*)
METHOD parse : BOOL
VAR_INPUT
	NMEAsentence : TNMEAsentence;
END_VAR
VAR_INST
	N 			: INT;
	msglen 		: INT;
	structlen	: INT;
	fieldtype	: BYTE;
	cbyte		: BYTE;
	fieldindex 	: INT;
	chkSumSentence  : USINT;
	chkSumCalc		: USINT;
	pbyte 			: POINTER TO BYTE; 
	ptypebyte		: POINTER TO BYTE;
	pbuffer 		: POINTER TO BYTE;
	pspointer		: POINTER TO STRING;
	buffer 			: TNMEAsentence;
END_VAR
parse := TRUE;
IF NOT getChkSumFromSentence(NMEAsentence, chkSumSentence) THEN
	parse := FALSE;
	RETURN;
END_IF

IF NOT calcChkSum(NMEASentence, chkSumCalc) THEN
	parse := FALSE;
	RETURN;
END_IF

IF chkSumCalc <> chkSumSentence THEN
	parse := FALSE;
	RETURN;
END_IF

msglen := len(NMEAsentence);
structlen := len(THIS^.sentenceStructure);

fieldindex := -1;

pbyte := ADR(NMEAsentence)+1;
ptypebyte := ADR(sentenceStructure);
pbuffer := ADR(buffer);

FOR N := 2 TO (msglen-2) DO
	cbyte := pbyte^;	
	
	CASE cbyte OF
		44, 42: // , and *
			pbuffer^ := 0;
			pbuffer := ADR(buffer); 
			pspointer := pbuffer;
			IF fieldindex = -1 THEN
				THIS^.header := pspointer^;
				fieldindex := 0;
			ELSE
				CASE ptypebyte^ OF
					73: // I
						THIS^.intFields[fieldindex] := STRING_TO_LINT(buffer);
						
					82: // R
						THIS^.realFields[fieldindex] := STRING_TO_LREAL(buffer);
						
					83: // S
					IF LEN(buffer) <= TNMEAstringsz THEN 
						THIS^.stringFields[fieldindex] := buffer;
					ELSE
						THIS^.stringFields[fieldindex] := '.';
					END_IF						
				END_CASE
				_incp(ptypebyte);
				fieldindex := fieldindex + 1;
				IF (structlen <= fieldindex) OR (cbyte = 42) THEN
					RETURN;
				END_IF
			END_IF
	ELSE
		pbuffer^ := cbyte;
		_incp(pbuffer);
 
	END_CASE	 
	_incp(pbyte);
 END_FOR
END_METHOD

(*
Purpose
=======
Set an string for field elements which are getting extracted. 
The position of a format char in the string is associated with the field number. 
The type of the field is given by the character

  I : Long Integer
  S : String(64)
  R : LReal
  . : Don't extract field
  
  Example:
  
  '..RR..I'
 
*)
METHOD setFieldsOfInterest : BOOL
VAR_INPUT
	Description : TNMEAStructDescription;
END_VAR
THIS^.sentenceStructure := Description;
END_METHOD

END_FUNCTION_BLOCK

// NMEA/NMEASentence
FUNCTION_BLOCK NMEASentence
VAR_INPUT
	
END_VAR
VAR
	formatString : FB_FormatString2;
	_dataOut : TNMEASentence;	
END_VAR

METHOD PROTECTED calcCheckSum : STRING
VAR_INPUT
	data : REFERENCE TO TNMEAsentence;	
END_VAR
VAR
	checksum : USINT;
	msglen : INT;
	N : INT;
	chksum : BYTE;
	char : BYTE; 
	pbyte : POINTER TO BYTE;
	x : BYTE;	
END_VAR
checksum := 0;
msglen := LEN(Data);
pbyte := ADR(data)+1;

FOR N := 2 TO msglen DO
	IF (pbyte^=42) THEN // Char *
		EXIT;
	ELSIF  (pbyte^=10) OR (pbyte^=13) THEN // Chars NL and CR
		EXIT;
	END_IF
	
	checksum := checksum XOR pbyte^;
	pbyte := pbyte + 1;
END_FOR

calcCheckSum :=  BYTE_TO_HEXSTR(In:= checksum, iPrecision:=2, bLoCase:=FALSE);
END_METHOD

PROPERTY DataOut : STRING
GET
DataOut := _dataout;
END_GET
END_PROPERTY

METHOD formatSentenceWith3Values : BOOL
VAR_INPUT
	NMEAType: REFERENCE TO T_MaxString;	
	Value1 	: LREAL;
	Value2 	: LREAL;
	Value3 	: LREAL;
END_VAR
VAR CONSTANT
		FORMATSTR 	: TNMEASentence := '%S,%.2F,%.2F,%.2F*  $0D$0A';
END_VAR
VAR
	checksum : STRING;
	datalen : INT;
END_VAR
formatString(pFormatString:=ADR(FORMATSTR), 
					arg1:=F_STRING(NMEAType), arg2:=F_LREAL(Value1), arg3:= F_LREAL(Value2), arg4:=F_LREAL(Value3), 
					pDstString:=ADR(_dataOut), nDstSize:=TO_UDINT(255)); 
					
		
checksum := calcCheckSum(data:=_dataout);
datalen := LEN(_dataout);


_dataout := REPLACE(_dataout,checksum, 2, datalen-3);
END_METHOD

END_FUNCTION_BLOCK

// NMEA/NMEA_TrawlLength
FUNCTION_BLOCK NMEA_TrawlLength EXTENDS NMEASentence
VAR_INPUT
	LengthSTBD 	: LREAL;
	LengthPORT 	: LREAL;
	LengthMID 	: LREAL;	
END_VAR
VAR CONSTANT
	NMEAType : T_MaxString := '@TAWWL';
END_VAR

SUPER^.formatSentenceWith3Values(NMEAType:= NMEAType, Value1:=LengthSTBD, Value2:=LengthPORT, Value3:=LengthMID);

END_FUNCTION_BLOCK

// NMEA/NMEA_TrawlSpeed
FUNCTION_BLOCK NMEA_TrawlSpeed EXTENDS NMEASentence
VAR_INPUT
	SpeedSTBD 	: LREAL;
	SpeedPORT 	: LREAL;
	SpeedMID 	: LREAL;	
END_VAR
VAR CONSTANT
	NMEAType : T_MaxString := '@TAWWS';
END_VAR

VAR_OUTPUT
END_VAR
VAR
END_VAR

SUPER^.formatSentenceWith3Values(NMEAType:= NMEAType, Value1:=SpeedSTBD, Value2:=SpeedPORT, Value3:=SpeedMID);

END_FUNCTION_BLOCK

// NMEA/NMEA_TrawlTension
FUNCTION_BLOCK NMEA_TrawlTension EXTENDS NMEASentence
VAR_INPUT
	TensionSTBD 	: LREAL;
	TensionPORT 	: LREAL;
	TensionMID 	: LREAL;	
END_VAR
VAR CONSTANT
	NMEAType : T_MaxString := '@TAWWT';
END_VAR

VAR_OUTPUT
END_VAR
VAR
END_VAR

SUPER^.formatSentenceWith3Values(NMEAType:= NMEAType, Value1:=TensionSTBD, Value2:=TensionPORT, Value3:=TensionMID);

END_FUNCTION_BLOCK

// NMEA/NMEATransmitter6021
FUNCTION_BLOCK NMEATransmitter6021
VAR_INPUT
	data 	: REFERENCE TO TNMEASentence;
	start   : BOOL;
END_VAR
VAR
	dataout AT %Q*  : ARRAY[0..97] OF BYTE;
	sword	AT %I*  : WORD;
	cword	AT %Q*  : WORD;
	_busy			: BOOL;
	state			: DINT;
	started			: BOOL;
END_VAR



CASE state OF
	0: 
		_busy := FALSE;
		IF NOT started THEN
			state := 100;
		ELSIF start THEN
			state := 10;
		END_IF
	10:
		_busy := TRUE;
		strncpy(ADR(dataout), ADR(data), TO_UINT(LEN(data)+1));
		cword := SHL(TO_UINT(len(data)), 8) OR (cword AND 16#0001);
		cword.0 := NOT cword.0;
		_busy := TRUE;
		state := 20;
		
	20:
		IF sword.0 THEN
			state := 0;
		END_IF
	
	100:
		_busy := TRUE;
		cword.2 := TRUE;	
		IF sword.2 AND NOT start THEN
			cword.2 := FALSE;
			started :=TRUE;
			state := 110; 
		END_IF	
		
	110: 
		cword := 0;
		IF NOT sword.2	THEN
			state := 0;
			_busy := FALSE;
		END_IF
END_CASE

PROPERTY Busy : BOOL
GET
Busy := _busy;
END_GET
END_PROPERTY

END_FUNCTION_BLOCK

// ObjectProtocols/V1/ProtoBase1ToN
(* 
Protocol Base Class 1:N
=======================

The class is class partially implementing a simple relation between objects of 1:N

This class has to be derived and can't be used out of the box. 

You have to take care of _noElements, _totalSize

*)

{attribute 'hide_all_locals'}
FUNCTION_BLOCK ABSTRACT ProtoBase1ToN IMPLEMENTS p7type.IProtoBase1ToN
VAR
	_noElements : DINT;
	_totalSize  : DINT;
END_VAR

METHOD attach : IProtoBase1ToN
VAR_INPUT
	Service : IProtoService;
END_VAR
VAR
	N	 		: DINT;
	_service	: IProtoService;
END_VAR

FOR N := 0 TO THIS^._totalSize-1 DO
	//We can't compare an Interface value returned from a method, which makes this 
	// necessary
	_service := getService(N);
	IF _service = Service THEN
		EXIT;
	ELSIF _service = 0 THEN
		setService(N, Service);
		_noElements := _noElements + 1;
		EXIT;
	END_IF
END_FOR

attach := THIS^;
END_METHOD

// This method has initialize _totalSize
METHOD FB_init : BOOL
VAR_INPUT
	bInitRetains : BOOL; // if TRUE, the retain variables are initialized (warm start / cold start)
	bInCopyCode : BOOL;  // if TRUE, the instance afterwards gets moved into the copy code (online change)
END_VAR
THIS^._totalSize := Parameters.ServicesPerMaster;

_noElements := 0;
END_METHOD

METHOD getNoServices : DINT
getNoServices := _noElements;
END_METHOD

// Overwrite this method
METHOD PROTECTED ABSTRACT getService : IProtoService
VAR_INPUT
	Index  : DINT;
END_VAR
END_METHOD

METHOD getServiceByIdx : IProtoService
VAR_INPUT
	Index  : DINT;
END_VAR
getServiceByIdx := getService(Index);
END_METHOD

METHOD isAttached : BOOL
VAR_INPUT
	Service : IProtoService;
END_VAR
VAR
	N : DINT;
	_service	: IProtoService;
END_VAR
isAttached := FALSE;
FOR N := 0 TO THIS^._totalSize-1 DO
	//We can't compare an Interface value returned from a method, which makes this 
	// necessary
	_service := getService(N);
	IF Service = _service THEN
		isAttached := TRUE;
		EXIT;
	ELSIF _service = 0 THEN
		EXIT;
	END_IF
END_FOR
END_METHOD

METHOD resetService : IProtoBase1ToN
VAR
	N 			: DINT;
	noElements 	: DINT;
END_VAR
FOR N := 0 TO THIS^._totalSize-1 DO
	setService(N, 0);
END_FOR

THIS^._noElements := 0;

resetService := THIS^;
END_METHOD

// Overwrite this method
METHOD PROTECTED ABSTRACT setService : IProtoBase1ToN
VAR_INPUT
	Index : DINT;
	Value : IProtoService;
END_VAR
END_METHOD

END_FUNCTION_BLOCK

// ObjectProtocols/V1/ProtoBaseNTo1
(* 
Protocol Base Class N:1
=======================

The class is class partially implementing a simple relation between objects of N:1. The 1 element is a master, which 
has to provide IProtoMasterSingleService to attach remote a Service by the service

This class has to be derived and can't be used out of the box. 

You have to take care of _noElements, _totalSize


*)

{attribute 'hide_all_locals'}
FUNCTION_BLOCK ABSTRACT ProtoBaseNTo1 IMPLEMENTS p7type.IProtoBaseNTo1
VAR
	_noElements : DINT;
	_totalSize  : DINT;
END_VAR

METHOD attach : IProtoBaseNTo1
VAR_INPUT
	Master	: IProtoMasterSingleService;
END_VAR
VAR
	N 		: DINT;
	_master : IProtoMasterSingleService;
END_VAR

FOR N := 0 TO THIS^._totalSize-1 DO
	_master := THIS^.getMaster(N);
	IF _master = Master THEN
		EXIT;
	ELSIF _master = 0 THEN
		setMaster(N, Master);
		Master.attach(THIS^);
		_noElements := _noElements + 1;
		EXIT;
	END_IF
END_FOR

attach := THIS^;
END_METHOD

// This method has initialize _totalSize
METHOD FB_init : BOOL
VAR_INPUT
	bInitRetains : BOOL; // if TRUE, the retain variables are initialized (warm start / cold start)
	bInCopyCode : BOOL;  // if TRUE, the instance afterwards gets moved into the copy code (online change)
END_VAR
THIS^._totalSize := Parameters.MastersPerService;

_noElements := 0;
END_METHOD

{attribute 'monitoring' := 'call'}
// Overwrite this method
METHOD PROTECTED ABSTRACT getMaster : IProtoMasterSingleService
VAR_INPUT
	Index  : DINT;
END_VAR
END_METHOD

METHOD getMasterByIdx : IProtoMasterSingleService
VAR_INPUT
	Index  : DINT;
END_VAR
	getMasterByIdx := getMaster(Index);
END_METHOD

METHOD getNoMasters : DINT
getNoMasters := THIS^._noElements;
END_METHOD

METHOD isAttached : BOOL
VAR_INPUT
	Master	: IProtoMasterSingleService;
END_VAR
VAR
	N : DINT;
	_master : IProtoMasterSingleService;
END_VAR
isAttached := FALSE;
FOR N := 0 TO THIS^._totalSize-1 DO
	_master := getMaster(N);
	IF Master = _master THEN
		isAttached := TRUE;
		EXIT;
	ELSIF _master = 0 THEN
		EXIT;
	END_IF
END_FOR
END_METHOD

METHOD resetServices : IProtoBaseNTo1
VAR
	N : DINT;
END_VAR
FOR N := 0 TO _totalSize-1 DO
	setMaster(N, 0);
END_FOR
_noElements := 0;

resetServices := THIS^;
END_METHOD

// Overwrite this method
METHOD PROTECTED setMaster : IProtoBaseNTo1
VAR_INPUT
	Index : DINT;
	Value : IProtoMasterSingleService;
END_VAR
END_METHOD

END_FUNCTION_BLOCK

// ObjectProtocols/V1/ProtoMasterSingleService

{attribute 'hide_all_locals'}
FUNCTION_BLOCK ProtoMasterSingleService IMPLEMENTS p7type.IProtoMasterSingleService
VAR
	service 			: IProtoService; 
END_VAR

METHOD attach : IProtoMasterSingleService
VAR_INPUT
	Service	: IProtoService;
END_VAR
THIS^.service := Service;

attach := THIS^;
END_METHOD

METHOD getService : IProtoService
getService := THIS^.service;
END_METHOD

END_FUNCTION_BLOCK

// OperationTime/DeviceOpTime
(* This utility class is counting optime for winches in hours
	Internaly the counter is of type TIME, but the output is of type UINT
*)
FUNCTION_BLOCK DeviceOpTime
VAR_INPUT
	Device : p7type.IP6OpState;
END_VAR
VAR PERSISTENT
	_optime : TIME;
END_VAR
VAR
	counter : OperationTimeCounter;
END_VAR

IF Device = 0 THEN
	RETURN;
END_IF

counter.update(
	active := Device.OpState = p7type.P6OpState.RUN,
	operationTime := _optime
);

{attribute 'monitoring' := 'call'}
{attribute 'TcRpcEnable'}
PROPERTY Optime : UDINT
GET
OpTime := TIME_TO_UDINT(_optime/UDINT#3600000);
END_GET
SET
_optime := UDINT_TO_TIME(Optime*UDINT#3600000);
END_SET
END_PROPERTY

END_FUNCTION_BLOCK

// OperationTime/OperationTimeCounter
// The class measures the active-time and adds it to the referenced operationTime. 
{attribute 'hide_all_locals'}
FUNCTION_BLOCK OperationTimeCounter
VAR
	_startTime 			: TIME;
	_state 				: OperationTimeSM;
	optime				: REFERENCE TO TIME;
END_VAR

METHOD reset : BOOL
THIS^.optime := T#0S;
END_METHOD

METHOD update : BOOL
VAR_INPUT
	active : BOOL;
	operationTime : REFERENCE TO TIME;
END_VAR
optime REF= operationTime;

CASE _state OF
	OperationTimeSM.IDLE:
		IF active THEN
			_state := OperationTimeSM.ACTIVE;
			_startTime := TIME();
		END_IF
			
	OperationTimeSM.ACTIVE:
		IF NOT active THEN
			operationTime := operationTime + (TIME() - _startTime);
			_state := OperationTimeSM.IDLE;
		ELSE
			_state := OperationTimeSM.ACTIVE;
			operationTime := operationTime + (TIME() - _startTime);
			_startTime := TIME();			
		END_IF
END_CASE
END_METHOD

END_FUNCTION_BLOCK

// ParameterManagment/AddParameter/AddParameterBool
FUNCTION_BLOCK AddParameterBool
VAR_INPUT
	parameterName : STRING := 'NoParameterNameSet'; //Parameter name to be displayed
	unit : STRING := ''; //SI units (m, kg, Nm, etc.)
	uploadParameter : BOOL := FALSE; //Update parameters to PLC
	downloadParameter : BOOL := FALSE; //Download parameters to HMI
END_VAR
VAR_OUTPUT
END_VAR
VAR_IN_OUT
	configMember : BOOL;
	parameterList : ParameterList;
END_VAR
VAR
	_init : BOOL := TRUE;
END_VAR

IF _init THEN
	_init := FALSE;
	parameterList.name := parameterName;
	parameterList.unit := unit;
END_IF

IF uploadParameter THEN
	configMember := parameterList.value.boolType;
END_IF

IF downloadParameter THEN
	parameterList.value.boolType := configMember;
END_IF

//Check status on parameter between config and parameter list
IF (parameterList.value.boolType = configMember)
THEN
	parameterList.status := 'Ok';
ELSE
	parameterList.status := 'Missmatch!';
END_IF

END_FUNCTION_BLOCK

// ParameterManagment/AddParameter/AddParameterInt
FUNCTION_BLOCK AddParameterInt
VAR_INPUT
	parameterName : STRING := 'NoParameterNameSet'; //Parameter name to be displayed
	unit : STRING := ''; //SI units (m, kg, Nm, etc.)
	uploadParameter : BOOL := FALSE; //Update parameters to PLC
	downloadParameter : BOOL := FALSE; //Download parameters to HMI
END_VAR
VAR_OUTPUT
END_VAR
VAR_IN_OUT
	configMember : INT;
	parameterList : ParameterList;
END_VAR
VAR
	_init : BOOL := TRUE;
END_VAR

IF _init THEN
	_init := FALSE;
	parameterList.name := parameterName;
	parameterList.unit := unit;
END_IF

IF uploadParameter THEN
	configMember := parameterList.value.intType;
END_IF

IF downloadParameter THEN
	parameterList.value.intType := configMember;
END_IF

//Check status on parameter between config and parameter list
IF (parameterList.value.intType = configMember)
THEN
	parameterList.status := 'Ok';
ELSE
	parameterList.status := 'Missmatch!';
END_IF

END_FUNCTION_BLOCK

// ParameterManagment/AddParameter/AddParameterLreal
FUNCTION_BLOCK AddParameterLreal
VAR_INPUT
	parameterName : STRING := 'NoParameterNameSet'; //Parameter name to be displayed
	unit : STRING := ''; //SI units (m, kg, Nm, etc.)
	uploadParameter : BOOL := FALSE; //Update parameters to PLC
	downloadParameter : BOOL := FALSE; //Download parameters to HMI
END_VAR
VAR_OUTPUT
END_VAR
VAR_IN_OUT
	configMember : LREAL;
	parameterList : ParameterList;
END_VAR
VAR
	_init : BOOL := TRUE;
END_VAR

IF _init THEN
	_init := FALSE;
	parameterList.name := parameterName;
	parameterList.unit := unit;
END_IF

IF uploadParameter THEN
	configMember := parameterList.value.lrealType;
END_IF

IF downloadParameter THEN
	parameterList.value.lrealType := configMember;
END_IF

//Check status on parameter between config and parameter list
IF (parameterList.value.lrealType = configMember)
THEN
	parameterList.status := 'Ok';
ELSE
	parameterList.status := 'Missmatch!';
END_IF

END_FUNCTION_BLOCK

// ParameterManagment/AddParameter/AddParameterStr
FUNCTION_BLOCK AddParameterStr
VAR_INPUT
	parameterName : STRING := 'NoParameterNameSet'; //Parameter name to be displayed
	unit : STRING := ''; //SI units (m, kg, Nm, etc.)
	uploadParameter : BOOL := FALSE; //Update parameters to PLC
	downloadParameter : BOOL := FALSE; //Download parameters to HMI
END_VAR
VAR_OUTPUT
END_VAR
VAR_IN_OUT
	configMember : STRING;
	parameterList : ParameterList;
END_VAR
VAR
	_init : BOOL := TRUE;
END_VAR

IF _init THEN
	_init := FALSE;
	parameterList.name := parameterName;
	parameterList.unit := unit;
END_IF

IF uploadParameter THEN
	configMember := parameterList.value.stringType;
END_IF

IF downloadParameter THEN
	parameterList.value.stringType := configMember;
END_IF

//Check status on parameter between config and parameter list
IF (parameterList.value.stringType = configMember)
THEN
	parameterList.status := 'Ok';
ELSE
	parameterList.status := 'Missmatch!';
END_IF

END_FUNCTION_BLOCK

// ParameterManagment/AddParameter/AddParameterTime
FUNCTION_BLOCK AddParameterTime
VAR_INPUT
	parameterName : STRING := 'NoParameterNameSet'; //Parameter name to be displayed
	unit : STRING := ''; //SI units (m, kg, Nm, etc.)
	uploadParameter : BOOL := FALSE; //Update parameters to PLC
	downloadParameter : BOOL := FALSE; //Download parameters to HMI
END_VAR
VAR_OUTPUT
END_VAR
VAR_IN_OUT
	configMember : TIME;
	parameterList : ParameterList;
END_VAR
VAR
	_init : BOOL := TRUE;
	_msPerSecond : LREAL := 1000.0;
END_VAR

IF _init THEN
	_init := FALSE;
	parameterList.name := parameterName;
	parameterList.unit := unit;
END_IF

IF uploadParameter THEN
	configMember := LREAL_TO_TIME(parameterList.value.lrealType * _msPerSecond);
END_IF

IF downloadParameter THEN
	parameterList.value.lrealType := TIME_TO_LREAL(configMember) / _msPerSecond;
END_IF

//Check status on parameter between config and parameter list
IF (parameterList.value.lrealType * _msPerSecond = TIME_TO_LREAL(configMember)) THEN
	parameterList.status := 'Ok';
ELSE
	parameterList.status := 'Missmatch!';
END_IF

END_FUNCTION_BLOCK

// PID/HTrawlController
(*
Purpose
=======
This is a 2 stage P-PI controller for trawling withg hydraulic winches.
This is the first version and only for documentations purposes in this lib. 

Features
========
#. This version has no stepped P controller for velocity
#. Anti Windup for the integrator
#. Symmetric processing to 0 of input values
#. Limiting output values 

Methods And Properties
======================
*)
{attribute 'hide_all_locals'}
FUNCTION_BLOCK HTrawlController;
VAR_INPUT
	config 				: REFERENCE TO p7type.ConfigTrawlController;
	Active 				: BOOL;		
	IsInRun				: BOOL;
	PayoutMode			: BOOL;
	Setpoint 			: LREAL;	// Length setpoint
	ProcessValueLen		: LREAL;	// Length process value
	ProcessValueVel		: LREAL;	// Velocity process value
	ProcessValueTension : LREAL;	// Tension process value 
	ProcessValueTorqueRel: LREAL;
	LimitVel			: LREAL;
	LimitTensionMax		: LREAL;
	LimitTensionMin		: LREAL;
	LimitTorqueRelMax	: LREAL;
	LimitTorqueRelMin	: LREAL;
	IntegratorPresetRel : LREAL;
	ReduceEnergyUsage	: BOOL;
	CycleTime			: LREAL;
END_VAR
VAR CONSTANT
	ALMOST_ZERO 		: LREAL := 1.0/60.0;
END_VAR
VAR
	startTrig 			: R_TRIG;
	_torqueOut 			: LREAL;
	Tc					: LREAL;
	errorLen			: LREAL;
	errorVel			: LREAL;
	deltaIt				: LREAL;
	tmp 				: LREAL;
	It					: LREAL;
	Pt					: LREAL;
	
	setpointVelocity		: LREAL;
	step				: DINT;
	velocityReduction   : LREAL;
	timerReducePower	: BOOL;
	statePos			: UINT;
	positionChange		: BOOL;
	offsetTension		: LREAL;
	pValueTension		: LREAL;
	pLimitTensionMax	: LREAL;
	pLimitTensionMin	: LREAL;
END_VAR

Tc := CycleTime;
//
// Process the position error
// 
errorLen :=  (SetPoint - ProcessValueLen);
 
(* Process deadband *)
IF Config.DeadbandLength > 0 THEN
	IF (ABS(errorLen) < (Config.DeadbandLength/2.0)) THEN
		errorLen := 0.0;
	ELSE 
		errorLen := errorLen - Signum(errorLen) * Config.DeadbandLength/2.0; 
	END_IF;
END_IF;

IF Active THEN
	// Initiatlize integrator for torque
	startTrig(CLK:=Active);
	IF startTrig.Q AND IsInRun THEN
		It := ProcessValueTorqueRel-0.5;
		step := 0;
	ELSIF startTrig.Q AND (NOT IsInRun)  THEN
		It :=  LIMIT(-0.5, IntegratorPresetRel-0.5, 0.5);
	END_IF
		
	IF ReduceEnergyUsage THEN 
		velocityReduction := 0.1;
	ELSE
		velocityReduction := 1;
	END_IF
	setpointVelocity := LIMIT(-LimitVel*velocityReduction ,errorLen*config.KpVelocity*velocityReduction, LimitVel*velocityReduction);
	//setpointVelocity := LIMIT(-LimitVel ,errorLen * config.KpVelocity, LimitVel);
	
	//
	// Tension controller -> Control velocity with torque
	//

	// The minus has to be used bc of torque has the opposite direction to velocity 
	errorVel := - (setpointVelocity - ProcessValueVel);	
	Pt := config.KpTorque * errorVel;
	
	
	IF ProcessValueVel <= (-LimitVel) THEN
		It := It - config.KiVelocityLimit;
		It := LIMIT(-0.5, It, 0.5);
		step := 2;
	ELSIF ProcessValueVel >= (LimitVel) THEN
		It := It + config.KiVelocityLimit;
		It := LIMIT(-0.5, It, 0.5);				
		step := 3;
	ELSIF (ProcessValueTension  < LimitTensionMin) THEN
		It := It + config.KiTensionLimit;
		It := LIMIT(-0.5, It, 0.5);
		step := 4;
	ELSIF (ProcessValueTension  > LimitTensionMax) AND (NOT PayoutMode) THEN
		It := It - config.KiTensionLimit;
		It := LIMIT(-0.5, It, 0.5);
		step := 5;
	ELSIF ABS(Config.KiTorque) <= 1E-100 THEN
		It :=  0.0;
		deltaIt := 0.0;
		step := 6;
	ELSE
		step := 1;
		// Start the check whether the new output would saturate and don't integrate when 
		// this is case
		deltaIt := errorVel * config.KiTorque * Tc;
		
		tmp := Pt + It + deltaIt;
		
		IF ABS(tmp) <= 0.5  THEN
			It := It + deltaIt;
		END_IF		
	END_IF

	
	_torqueOut := LIMIT(0, (Pt + It + 0.5), 1);	
ELSE
	_torqueOut := ProcessValueTorqueRel;// normalized to 1
END_IF;

{attribute 'TcRpcEnable'}
{attribute 'monitoring' := 'variable'}
PROPERTY ErrorPosition : LREAL
GET
ErrorPosition := errorLen;
END_GET
END_PROPERTY

{attribute 'TcRpcEnable'}
{attribute 'monitoring' := 'variable'}
PROPERTY ErrorVelocity : LREAL
GET
ErrorVelocity := errorVel;
END_GET
END_PROPERTY

{attribute 'TcRpcEnable'}
{attribute 'monitoring' := 'variable'}
PROPERTY Tension : LREAL
GET
Tension := TorqueOut;
END_GET
END_PROPERTY

PROPERTY TorqueOut : LREAL
GET
TorqueOut := _torqueOut;
END_GET
END_PROPERTY

END_FUNCTION_BLOCK

// PID/HTrawlController2
(*
Purpose
=======
This is a 2 stage P-PI controller for trawling withg hydraulic winches
This 2nd version is limit velocity via setpoint for the inner controller and
tension via limiting torqueRel. 

Features
========
#. This version has no stepped P controller for velocity
#. Anti Windup for the integrator
#. Symmetric processing to 0 of input values
#. Limiting output values 

Methods And Properties
======================
*)
{attribute 'hide_all_locals'}
FUNCTION_BLOCK HTrawlController2;
VAR_INPUT
	config 				: REFERENCE TO p7type.ConfigTrawlController;
	Active 				: BOOL;		
	IsInRun				: BOOL;
	PayoutMode			: BOOL;
	Setpoint 			: LREAL;	// Length setpoint
	ProcessValueLen		: LREAL;	// Length process value
	ProcessValueVel		: LREAL;	// Velocity process value
	ProcessValueTension : LREAL;	// Tension process value 
	ProcessValueTorqueRel: LREAL;
	LimitVel			: LREAL;
	LimitTensionMax		: LREAL;
	LimitTensionMin		: LREAL;
	LimitTorqueRelMax	: LREAL;
	LimitTorqueRelMin	: LREAL;
	IntegratorPresetRel : LREAL;
	ReduceEnergyUsage	: BOOL;
	CycleTime			: LREAL;
END_VAR
VAR CONSTANT
	ALMOST_ZERO 		: LREAL := 1.0/60.0;
END_VAR

VAR
	startTrig 			: R_TRIG;
	_torqueOut 			: LREAL;
	Tc					: LREAL;
	errorLen			: LREAL;
	errorVel			: LREAL;
	deltaIt				: LREAL;
	tmp 				: LREAL;
	It					: LREAL;
	Pt					: LREAL;
	
	setpointVelocity		: LREAL;
	step				: DINT;
	velocityReduction   : LREAL;
	timerReducePower	: BOOL;
	statePos			: UINT;
	positionChange		: BOOL;
	offsetTension		: LREAL;
	pValueTension		: LREAL;
	pLimitTensionMax	: LREAL;
	pLimitTensionMin	: LREAL;
	
END_VAR

Tc := CycleTime;
//
// Process the position error
// 
errorLen :=  (SetPoint - ProcessValueLen);
 
(* Process deadband *)
IF Config.DeadbandLength > 0 THEN
	IF (ABS(errorLen) < (Config.DeadbandLength/2.0)) THEN
		errorLen := 0.0;
	ELSE 
		errorLen := errorLen - Signum(errorLen) * Config.DeadbandLength/2.0; 
	END_IF;
END_IF;

startTrig(CLK:=Active);

IF Active THEN
	// Initiatlize integrator for torque
	IF startTrig.Q AND IsInRun THEN
		It := ProcessValueTorqueRel-0.5;
		step := 0;
	ELSIF startTrig.Q AND (NOT IsInRun)  THEN
		It :=  LIMIT(-0.5, IntegratorPresetRel-0.5, 0.5);
	END_IF
		
	
	IF ReduceEnergyUsage THEN
		step := 2; 
		velocityReduction := 0.1;
	ELSIF ProcessValueVel <= -LimitVel THEN
		step := 5; 
		velocityReduction := 0.0;
	ELSIF ProcessValueVel >= LimitVel THEN
		step := 6; 
		velocityReduction := 0.80;
	ELSE
		step := 1; 
		velocityReduction := 1;
	END_IF
	
	setpointVelocity := LIMIT(-LimitVel*velocityReduction ,errorLen*config.KpVelocity*velocityReduction, LimitVel*velocityReduction);

	//
	// Tension controller -> Control velocity with torque
	//

	// The minus has to be used bc of torque has the opposite direction to velocity 
	errorVel := - (setpointVelocity - ProcessValueVel);	
	Pt := config.KpTorque * errorVel;
	
	
	IF ABS(Config.KiTorque) <= 1E-100 THEN
		It :=  0.0;
		deltaIt := 0.0;
	ELSE
		// Start the check whether the new output would saturate and don't integrate when 
		// this is case
		deltaIt := errorVel * config.KiTorque * Tc;
		
		tmp := Pt + It + deltaIt;
		It := It + deltaIt;
		
		// integrate when between limits
		
		IF (tmp <= LimitTorqueRelMax-0.5) AND (tmp >= LimitTorqueRelMin-0.5)  THEN
			It := It + deltaIt;
		ELSIF (tmp < LimitTorqueRelMin - 0.5) THEN		
			It := (LimitTorqueRelMin-0.5 - Pt);
			step := 3;
		ELSIF (tmp > LimitTorqueRelMax - 0.5) THEN		
			It := (LimitTorqueRelMax - 0.5 - Pt);
			step := 4;
		END_IF		
	END_IF

	
	_torqueOut := LIMIT(0, (Pt + It + 0.5), 1);	
ELSE
	_torqueOut := ProcessValueTorqueRel;// normalized to 1
END_IF;

PROPERTY CtrlLimit : DINT
GET
CtrlLimit := Step;
END_GET
END_PROPERTY

{attribute 'TcRpcEnable'}
{attribute 'monitoring' := 'variable'}
PROPERTY ErrorPosition : LREAL
GET
ErrorPosition := errorLen;
END_GET
END_PROPERTY

{attribute 'TcRpcEnable'}
{attribute 'monitoring' := 'variable'}
PROPERTY ErrorVelocity : LREAL
GET
ErrorVelocity := errorVel;
END_GET
END_PROPERTY

{attribute 'TcRpcEnable'}
{attribute 'monitoring' := 'variable'}
PROPERTY Tension : LREAL
GET
Tension := TorqueOut;
END_GET
END_PROPERTY

PROPERTY TorqueOut : LREAL
GET
TorqueOut := _torqueOut;
END_GET
END_PROPERTY

PROPERTY VelocitySetpoint : LREAL
GET
VelocitySetpoint := setpointVelocity;
END_GET
END_PROPERTY

END_FUNCTION_BLOCK

// PID/HTrawlController3
(*
Purpose
=======
This is a 2 stage P-PI controller for trawling withg hydraulic winches
This 3. version is limiting Tension and Velocity via setpoint for the inner controller. 
 
Features
========
#. This version has no stepped P controller for velocity
#. Anti Windup for the integrator
#. Symmetric processing to 0 of input values
#. Limiting output values 

Methods And Properties
======================
*)
FUNCTION_BLOCK HTrawlController3;
VAR_INPUT
	config 				: REFERENCE TO p7type.ConfigTrawlController;
	Active 				: BOOL;		
	IsInRun				: BOOL;
	PayoutMode			: BOOL;
	Setpoint 			: LREAL;	// Length setpoint
	ProcessValueLen		: LREAL;	// Length process value
	ProcessValueVel		: LREAL;	// Velocity process value
	ProcessValueTension : LREAL;	// Tension process value 
	ProcessValueTorqueRel: LREAL;
	LimitVel			: LREAL;
	LimitTensionMax		: LREAL;
	LimitTensionMin		: LREAL;
	LimitTorqueRelMax	: LREAL;
	LimitTorqueRelMin	: LREAL;
	IntegratorPresetRel : LREAL;
	ReduceEnergyUsage	: BOOL;
	CycleTime			: LREAL;
END_VAR
VAR CONSTANT
	ALMOST_ZERO 		: LREAL := 1.0/60.0;
END_VAR

VAR
	startTrig 			: R_TRIG;
	_torqueOut 			: LREAL;
	Tc					: LREAL;
	errorLen			: LREAL;
	errorVel			: LREAL;
	deltaIt				: LREAL;
	tmp 				: LREAL;
	It					: LREAL;
	Pt					: LREAL;
	
	setpointVelocity		: LREAL;
	step				: DINT;
	velocityReduction   : LREAL;
	timerReducePower	: BOOL;
	statePos			: UINT;
	positionChange		: BOOL;
	offsetTension		: LREAL;
	pValueTension		: LREAL;
	pLimitTensionMax	: LREAL;
	pLimitTensionMin	: LREAL;
	
END_VAR

Tc := CycleTime;
//
// Process the position error
// 
errorLen :=  (SetPoint - ProcessValueLen);
 
(* Process deadband *)
IF Config.DeadbandLength > 0 THEN
	IF (ABS(errorLen) < (Config.DeadbandLength/2.0)) THEN
		errorLen := 0.0;
	ELSE 
		errorLen := errorLen - Signum(errorLen) * Config.DeadbandLength/2.0; 
	END_IF;
END_IF;

startTrig(CLK:=Active);

IF Active THEN
	// Initiatlize integrator for torque
	IF PayoutMode AND starttrig.Q THEN
		It := LIMIT(-0.5, IntegratorPresetRel-0.5, 0.5);
		It := ProcessValueTorqueRel-0.5;				
	ELSIF startTrig.Q AND IsInRun THEN
		It := ProcessValueTorqueRel-0.5;
		step := 0;
	ELSIF startTrig.Q AND (NOT IsInRun)  THEN
		It :=  LIMIT(-0.5, IntegratorPresetRel-0.5, 0.5);
	END_IF
		
	
	IF ReduceEnergyUsage THEN
		step := 2; 
		velocityReduction := 0.1;
	ELSIF (ProcessValueTension  > LimitTensionMax) AND (NOT PayoutMode) THEN 
		step := 3; 
		velocityReduction := 0;
	ELSIF (ProcessValueTension  < LimitTensionMin) THEN
		step := 4; 
		velocityReduction := 0;
	ELSIF ProcessValueVel <= -LimitVel THEN
		step := 5; 
		velocityReduction := 0;
	ELSIF ProcessValueVel >= LimitVel THEN
		step := 6; 
		velocityReduction := 0.50;
	ELSE
		step := 1; 
		velocityReduction := 1;
	END_IF
	
	setpointVelocity := LIMIT(-LimitVel*velocityReduction ,errorLen*config.KpVelocity*velocityReduction, LimitVel*velocityReduction);

	//
	// Tension controller -> Control velocity with torque
	//

	// The minus has to be used bc of torque has the opposite direction to velocity 
	errorVel := - (setpointVelocity - ProcessValueVel);	
	Pt := config.KpTorque * errorVel;
	
	
	IF ABS(Config.KiTorque) <= 1E-100 THEN
		It :=  0.0;
		deltaIt := 0.0;
	ELSE
		// Start the check whether the new output would saturate and don't integrate when 
		// this is case
		deltaIt := errorVel * config.KiTorque * Tc;
		
		tmp := Pt + It + deltaIt;
		// integrate when between limits
		IF ABS(tmp) <= 0.5  THEN
			It := It + deltaIt;
		END_IF		
	END_IF

	
	_torqueOut := LIMIT(0, (Pt + It + 0.5), 1);	
ELSE
	_torqueOut := ProcessValueTorqueRel;// normalized to 1
END_IF;

PROPERTY CtrlLimit : DINT
GET
CtrlLimit := Step;
END_GET
END_PROPERTY

{attribute 'TcRpcEnable'}
{attribute 'monitoring' := 'variable'}
PROPERTY ErrorPosition : LREAL
GET
ErrorPosition := errorLen;
END_GET
END_PROPERTY

{attribute 'TcRpcEnable'}
{attribute 'monitoring' := 'variable'}
PROPERTY ErrorVelocity : LREAL
GET
ErrorVelocity := errorVel;
END_GET
END_PROPERTY

{attribute 'TcRpcEnable'}
{attribute 'monitoring' := 'variable'}
PROPERTY Tension : LREAL
GET
Tension := TorqueOut;
END_GET
END_PROPERTY

PROPERTY TorqueOut : LREAL
GET
TorqueOut := _torqueOut;
END_GET
END_PROPERTY

PROPERTY VelocitySetpoint : LREAL
GET
VelocitySetpoint := setpointVelocity;
END_GET
END_PROPERTY

END_FUNCTION_BLOCK

// PID/HTrawlController4
(*
Purpose
=======
This is a 2 stage P-PI controller for trawling withg hydraulic winches
This 3. version is limiting Tension and Velocity via setpoint for the inner controller. 
 
Features
========
#. This version has no stepped P controller for velocity
#. Anti Windup for the integrator
#. Symmetric processing to 0 of input values
#. Limiting output values 

Methods And Properties
======================
*)
FUNCTION_BLOCK HTrawlController4;
VAR_INPUT
	config 				: REFERENCE TO p7type.ConfigTrawlController;
	Active 				: BOOL;		
	IsInRun				: BOOL;
	PayoutMode			: BOOL;
	HaulInMode			: BOOL;
	Setpoint 			: LREAL;	// Length setpoint
	ProcessValueLen		: LREAL;	// Length process value
	ProcessValueVel		: LREAL;	// Velocity process value
	ProcessValueTension : LREAL;	// Tension process value 
	ProcessValueTorqueRel: LREAL;
	LimitVel			: LREAL;
	LimitTensionMax		: LREAL;
	LimitTensionMin		: LREAL;
	LimitTorqueRelMax	: LREAL;
	LimitTorqueRelMin	: LREAL;
	IntegratorPresetRel : LREAL;
	ReduceEnergyUsage	: BOOL;
	CycleTime			: LREAL;
	VelStep1			: LREAL;
	VelStep2			: LREAL;
	VelStep3			: LREAL;
	VelStep4			: LREAL;
	VelStep5			: LREAL;
END_VAR
VAR CONSTANT
	ALMOST_ZERO 		: LREAL := 1.0/60.0;
END_VAR

VAR
	startTrig 			: R_TRIG;
	_torqueOut 			: LREAL;
	Tc					: LREAL;
	errorLen			: LREAL;
	errorVel			: LREAL;
	deltaIt				: LREAL;
	tmp 				: LREAL;
	It					: LREAL;
	Pt					: LREAL;
	
	setpointVelocity		: LREAL;
	step				: DINT;
	velocityReduction   : LREAL;
	timerReducePower	: BOOL;
	statePos			: UINT;
	positionChange		: BOOL;
	offsetTension		: LREAL;
	pValueTension		: LREAL;
	pLimitTensionMax	: LREAL;
	pLimitTensionMin	: LREAL;
	
END_VAR

Tc := CycleTime;
//
// Process the position error
// 
errorLen :=  (SetPoint - ProcessValueLen);
 
(* Process deadband *)
IF Config.DeadbandLength > 0 THEN
	IF (ABS(errorLen) < (Config.DeadbandLength/2.0)) THEN
		errorLen := 0.0;
	ELSE 
		errorLen := errorLen - Signum(errorLen) * Config.DeadbandLength/2.0; 
	END_IF;
END_IF;

startTrig(CLK:=Active);

IF Active THEN
	// Initiatlize integrator for torque
	IF PayoutMode AND starttrig.Q THEN
		It := ProcessValueTorqueRel-0.5;
	ELSIF startTrig.Q AND IsInRun THEN
		It := ProcessValueTorqueRel-0.5;
		step := 0;
	ELSIF startTrig.Q AND (NOT IsInRun)  THEN
		It :=  LIMIT(-0.5, IntegratorPresetRel-0.5, 0.5);
	END_IF
		
	
	IF ReduceEnergyUsage THEN
		step := 2; 
		velocityReduction := 0.1;
	ELSIF (ProcessValueTension  > LimitTensionMax) AND (NOT PayoutMode) THEN 
		step := 3; 
		velocityReduction := 0;
	ELSIF (ProcessValueTension  < LimitTensionMin) THEN
		step := 4; 
		velocityReduction := 0;
	ELSIF ProcessValueVel <= -LimitVel THEN
		step := 5; 
		velocityReduction := 0;
	ELSIF ProcessValueVel >= LimitVel THEN
		step := 6; 
		velocityReduction := 0.50;
	ELSE
		step := 1; 
		velocityReduction := 1;
	END_IF
	
	
	setpointVelocity := LIMIT(-LimitVel*velocityReduction ,errorLen*config.KpVelocity*velocityReduction, LimitVel*velocityReduction);

	IF PayoutMode OR HaulInMode THEN
		IF ABS(errorLen) < 1 AND ABS(setpointVelocity) > VelStep5 THEN
			setpointVelocity := VelStep5 * signum(setpointVelocity);
		ELSIF ABS(errorLen) < 5 AND ABS(setpointVelocity) > VelStep4 THEN
			setpointVelocity := VelStep4 * signum(setpointVelocity);
		ELSIF ABS(errorLen) < 10 AND ABS(setpointVelocity) > VelStep3 THEN
			setpointVelocity := VelStep3 * signum(setpointVelocity);
		ELSIF ABS(errorLen) < 15 AND ABS(setpointVelocity) > VelStep2 THEN
			setpointVelocity := VelStep2 * signum(setpointVelocity);
		ELSIF ABS(errorLen) < 20 AND ABS(setpointVelocity) > VelStep1 THEN
			setpointVelocity := VelStep1 * signum(setpointVelocity);				
		END_IF
	END_IF	
	
	//
	// Tension controller -> Control velocity with torque
	//

	// The minus has to be used bc of torque has the opposite direction to velocity 
	errorVel := - (setpointVelocity - ProcessValueVel);	
	Pt := config.KpTorque * errorVel;
	
	
	IF ABS(Config.KiTorque) <= 1E-100 THEN
		It :=  0.0;
		deltaIt := 0.0;
	ELSE
		// Start the check whether the new output would saturate and don't integrate when 
		// this is case
		deltaIt := errorVel * config.KiTorque * Tc;
		
		tmp := Pt + It + deltaIt;
		// integrate when between limits
		IF ABS(tmp) <= 0.5  THEN
			It := It + deltaIt;
		END_IF		
	END_IF

	
	_torqueOut := LIMIT(0, (Pt + It + 0.5), 1);	
ELSE
	_torqueOut := ProcessValueTorqueRel;// normalized to 1
END_IF;

PROPERTY CtrlLimit : DINT
GET
CtrlLimit := Step;
END_GET
END_PROPERTY

{attribute 'TcRpcEnable'}
{attribute 'monitoring' := 'variable'}
PROPERTY ErrorPosition : LREAL
GET
ErrorPosition := errorLen;
END_GET
END_PROPERTY

{attribute 'TcRpcEnable'}
{attribute 'monitoring' := 'variable'}
PROPERTY ErrorVelocity : LREAL
GET
ErrorVelocity := errorVel;
END_GET
END_PROPERTY

{attribute 'TcRpcEnable'}
{attribute 'monitoring' := 'variable'}
PROPERTY Tension : LREAL
GET
Tension := TorqueOut;
END_GET
END_PROPERTY

PROPERTY TorqueOut : LREAL
GET
TorqueOut := _torqueOut;
END_GET
END_PROPERTY

PROPERTY VelocitySetpoint : LREAL
GET
VelocitySetpoint := setpointVelocity;
END_GET
END_PROPERTY

END_FUNCTION_BLOCK

// PID/HTrawlController5
(*
Purpose
=======
This is a 2 stage P-PI controller for trawling withg hydraulic winches
This 3. version is limiting Tension and Velocity via setpoint for the inner controller. 
 
Features
========
#. This version has no stepped P controller for velocity
#. Anti Windup for the integrator
#. REMOVED: *** Symmetric processing to 0 of input values ***
#. Limiting output values 

Methods And Properties
======================
*)
FUNCTION_BLOCK HTrawlController5;
VAR_INPUT
	config 				: REFERENCE TO p7type.ConfigTrawlController;
	PrepareRegulator	: BOOL;		// store current torque value until active
	Active 				: BOOL;		// start command to activate auto
	IsInRun				: BOOL;		// currently always active from TrawlControl3
	PayoutMode			: BOOL;
	HaulInMode			: BOOL;
	Setpoint 			: LREAL;	// Length setpoint
	ProcessValueLen		: LREAL;	// Length process value
	ProcessValueVel		: LREAL;	// Velocity process value (m/s)
	ProcessValueTension : LREAL;	// Tension process value (Kg)
	ProcessValueTorqueRel: LREAL;	// 0-1 is full torque range
	LimitVel			: LREAL;	// highest speed allowed
	LimitTensionMax		: LREAL;	// highest tension allowed in tow or haul (kg)
	LimitTensionMin		: LREAL;	// lowest tension allowed in tow or pay (kg)
	LimitTorqueRelMax	: LREAL;	// highest torque allowed in tow or haul
	LimitTorqueRelMin	: LREAL;	// lowest torque allowed in tow or pay
	IntegratorPresetRel : LREAL;	// Initial value to use if winch is in stop (?)
	ReduceEnergyUsage	: BOOL;
	CycleTime			: LREAL;	// cycle time in s (usually 0.05)
	VelStep1			: LREAL;
	VelStep2			: LREAL;
	VelStep3			: LREAL;
	VelStep4			: LREAL;
	VelStep5			: LREAL;
END_VAR
VAR CONSTANT
	ALMOST_ZERO 		: LREAL := 1.0/60.0;
END_VAR

VAR
	saveTorque			: R_TRIG;		// store tension until regulator starts
	startTrig 			: R_TRIG;		// first scan after regulator is activated
	_torqueOut 			: LREAL;
	Tc					: LREAL;		// cycle time in s (usually 0.05)
	errorLen			: LREAL;		// distance from setpoint (positive is too long)
	errorVel			: LREAL;		// negative when too long (negated)
	deltaIt				: LREAL;		// Current interation's contribution to It 
	tmp 				: LREAL;
	It					: LREAL;		// integrator value
	Pt					: LREAL;		// proportional value
	
	initialTorqueRel	: LREAL;	// saved torque while waiting for regulator to start
	setpointVelocity	: LREAL;
	step				: DINT;
	velocityReduction   : LREAL;		// Used as a multiplicand to reduce velocity setpoint when limiting speed or torque
	timerReducePower	: BOOL;
	statePos			: UINT;
	positionChange		: BOOL;
	offsetTension		: LREAL;
	pValueTension		: LREAL;
	pLimitTensionMax	: LREAL;
	pLimitTensionMin	: LREAL;
	VelocityIsOverSetpoint	: BOOL;		// used to prevent further integration of Ki
	setpointVel_m_min	: LREAL;		// monitoring setpoint (meter/min)
	processVel_m_min	: LREAL;		// monitoring actual velocity (meter/min)
	lengthAtVelMax		: LREAL;		// monitoring: At which errorLength will setpointVel be at max? 
END_VAR

Tc := CycleTime;
//
// Process the position error
// 
errorLen :=  (SetPoint - ProcessValueLen);
 
(* Process deadband *)
IF Config.DeadbandLength > 0 THEN
	IF (ABS(errorLen) < (Config.DeadbandLength/2.0)) THEN
		errorLen := 0.0;
	ELSE 
		errorLen := errorLen - Signum(errorLen) * Config.DeadbandLength/2.0; 
	END_IF;
END_IF;

saveTorque(CLK := PrepareRegulator);
startTrig(CLK:=Active);

// store ProcessValueTorqueRel
IF saveTorque.Q THEN
	initialTorqueRel := ProcessValueTorqueRel;
END_IF

IF Active THEN
	// Initiatlize integrator for torque
	
	// removed, identical to next IF: 
	//IF PayoutMode AND starttrig.Q THEN
	//	It := ProcessValueTorqueRel;  //   -0.5;
	IF startTrig.Q AND IsInRun THEN
		It := initialTorqueRel; //   start the regulator with stored value
		step := 0;
	//currently as long as IsInRun is always true (see TrawlControl3), this will never run.
	ELSIF startTrig.Q AND (NOT IsInRun)  THEN
		It :=  LIMIT(0, IntegratorPresetRel, 1);  //LIMIT(-0.5, IntegratorPresetRel-0.5, 0.5);
	END_IF
	
	// set bit if haul in speed is too high
	VelocityIsOverSetpoint := SEL(ProcessValueVel <= -LimitVel,FALSE,TRUE);
	
	// limiting modes
	IF ReduceEnergyUsage THEN							// power consumed or regen too high
		step := 2; 
		velocityReduction := 0.3;
	ELSIF (ProcessValueTension  > LimitTensionMax) AND (NOT PayoutMode) THEN //too high tension (not payout)
		step := 3; 
		velocityReduction := 0.3;
	ELSIF (ProcessValueTension  < LimitTensionMin) THEN //too low tension
		step := 4; 
		velocityReduction := 0.3;
	ELSIF ProcessValueVel <= -LimitVel THEN		// haul in too fast
		step := 5; 					
		velocityReduction := 0.3;
	ELSIF ProcessValueVel >= LimitVel THEN		//pay out too fast
		step := 6; 
		velocityReduction := 0.50;
	ELSE										// everything's normal
		step := 1; 
		velocityReduction := 1;
	END_IF
	
	// KpVelocity: 20m error length and kp of 0.1 will give a setpointVelocity of 2 m/s or 120m/min
	// if LimitVel is active, limits and error length will be desimated accordingly limiting the setpointVelocity.
	setpointVelocity := LIMIT(-LimitVel*velocityReduction ,errorLen*config.KpVelocity*velocityReduction, LimitVel*velocityReduction);

	IF PayoutMode OR HaulInMode THEN
		IF ABS(errorLen) < 1 AND ABS(setpointVelocity) > VelStep5 THEN
			setpointVelocity := VelStep5 * signum(setpointVelocity);
		ELSIF ABS(errorLen) < 5 AND ABS(setpointVelocity) > VelStep4 THEN
			setpointVelocity := VelStep4 * signum(setpointVelocity);
		ELSIF ABS(errorLen) < 10 AND ABS(setpointVelocity) > VelStep3 THEN
			setpointVelocity := VelStep3 * signum(setpointVelocity);
		ELSIF ABS(errorLen) < 15 AND ABS(setpointVelocity) > VelStep2 THEN
			setpointVelocity := VelStep2 * signum(setpointVelocity);
		ELSIF ABS(errorLen) < 20 AND ABS(setpointVelocity) > VelStep1 THEN
			setpointVelocity := VelStep1 * signum(setpointVelocity);				
		END_IF
	END_IF	
	
	// calculate at which length the setpointVel is equal to limitVel
	// only used for monitoring
	lengthAtVelMax := (LimitVel / config.KpVelocity);
	processVel_m_min := ProcessValueVel * 60 ;
	setpointVel_m_min := setpointVelocity * 60 ;
	//
	// Tension controller -> Control velocity with torque
	//

	// The minus has to be used bc of torque has the opposite direction to velocity 
	errorVel := - (setpointVelocity - ProcessValueVel);	
	
	// If error velocity is 1 (60m) and KpTorque is 0.05 the output (Pt) will add  5% to the output signal
	
	Pt := config.KpTorque * errorVel;
	
	
	IF ABS(Config.KiTorque) <= 1E-100 THEN
		It :=  0.0;
		deltaIt := 0.0;
	ELSE
		// Start the check whether the new output would saturate and don't integrate when 
		// this is case
		// A KiTorque of 0.005 and errorVel of 1 (60 m/min) will increase regulator output with 0.5% per second
		deltaIt := errorVel * config.KiTorque * Tc;
	
		tmp := Pt + It + deltaIt;
		
		// integrate when between limits
		IF ABS(tmp) <= 1  THEN		// removed 0.5 - set to '1'
			It := It + deltaIt;
		END_IF		
	END_IF

	
	_torqueOut := LIMIT(0, (Pt + It), 1);  // +0.5 removed	

ELSIF PrepareRegulator THEN
	// auto is on its way, but not active yet
	_torqueOut := initialTorqueRel ;
ELSE
	// no auto function active
	_torqueOut := ProcessValueTorqueRel;// normalized to 1
END_IF;

PROPERTY CtrlLimit : DINT
GET
CtrlLimit := Step;
END_GET
END_PROPERTY

{attribute 'TcRpcEnable'}
{attribute 'monitoring' := 'variable'}
PROPERTY ErrorPosition : LREAL
GET
ErrorPosition := errorLen;
END_GET
END_PROPERTY

{attribute 'TcRpcEnable'}
{attribute 'monitoring' := 'variable'}
PROPERTY ErrorVelocity : LREAL
GET
ErrorVelocity := errorVel;
END_GET
END_PROPERTY

{attribute 'TcRpcEnable'}
{attribute 'monitoring' := 'variable'}
PROPERTY Tension : LREAL
GET
Tension := TorqueOut;
END_GET
END_PROPERTY

PROPERTY TorqueOut : LREAL
GET
TorqueOut := _torqueOut;
END_GET
END_PROPERTY

PROPERTY VelocitySetpoint : LREAL
GET
VelocitySetpoint := setpointVelocity;
END_GET
END_PROPERTY

END_FUNCTION_BLOCK

// PID/HTrawlController6
(*
Purpose
=======
This is a 2 stage P-PI controller for trawling withg hydraulic winches
This 3. version is limiting Tension and Velocity via setpoint for the inner controller. 
 
Features
========
#. This version has no stepped P controller for velocity
#. Anti Windup for the integrator
#. REMOVED: *** Symmetric processing to 0 of input values ***
#. Limiting output values 

Methods And Properties
======================
*)
FUNCTION_BLOCK HTrawlController6;
VAR_INPUT
	config 				: REFERENCE TO p7type.ConfigTrawlController;
	PrepareRegulator	: BOOL;		// store current torque value until active
	Active 				: BOOL;		// start command to activate auto
	IsInRun				: BOOL;		// currently always active from TrawlControl3
	PayoutMode			: BOOL;
	HaulInMode			: BOOL;
	Setpoint 			: LREAL;	// Length setpoint
	ProcessValueLen		: LREAL;	// Length process value
	ProcessValueVel		: LREAL;	// Velocity process value (m/s)
	ProcessValueTension : LREAL;	// Tension process value (Kg)
	ProcessValueTorqueRel: LREAL;	// 0-1 is full torque range
	LimitVel			: LREAL;	// highest speed allowed
	LimitTensionMax		: LREAL;	// highest tension allowed in tow or haul (kg)
	LimitTensionMin		: LREAL;	// lowest tension allowed in tow or pay (kg)
	LimitTorqueRelMax	: LREAL;	// highest torque allowed in tow or haul
	LimitTorqueRelMin	: LREAL;	// lowest torque allowed in tow or pay
	IntegratorPresetRel : LREAL;	// Initial value to use if winch is in stop (?)
	ReduceEnergyUsage	: BOOL;
	CycleTime			: LREAL;	// cycle time in s (usually 0.05)
	VelStep1			: LREAL;
	VelStep2			: LREAL;
	VelStep3			: LREAL;
	VelStep4			: LREAL;
	VelStep5			: LREAL;
	Freeze				: BOOL; // If true then simpelten route toqueRel to output
END_VAR
VAR CONSTANT
	ALMOST_ZERO 		: LREAL := 1.0/60.0;
END_VAR

VAR
	saveTorque			: R_TRIG;		// store tension until regulator starts
	startTrig 			: R_TRIG;		// first scan after regulator is activated
	_torqueOut 			: LREAL;
	Tc					: LREAL;		// cycle time in s (usually 0.05)
	errorLen			: LREAL;		// distance from setpoint (positive is too long)
	errorVel			: LREAL;		// negative when too long (negated)
	deltaIt				: LREAL;		// Current interation's contribution to It 
	tmp 				: LREAL;
	It					: LREAL;		// integrator value
	Pt					: LREAL;		// proportional value
	
	initialTorqueRel	: LREAL;	// saved torque while waiting for regulator to start
	setpointVelocity	: LREAL;
	step				: DINT;
	velocityReduction   : LREAL;		// Used as a multiplicand to reduce velocity setpoint when limiting speed or torque
	timerReducePower	: BOOL;
	statePos			: UINT;
	positionChange		: BOOL;
	offsetTension		: LREAL;
	pValueTension		: LREAL;
	pLimitTensionMax	: LREAL;		// do not allow output to go LOWER trhan this value
	pLimitTensionMin	: LREAL;		// do not allow output to go HIGHER trhan this value
	HaulInVelocityIsOverSetpoint	: BOOL;		// used to prevent further integration of Ki
	setpointVel_m_min	: LREAL;		// monitoring setpoint (meter/min)
	processVel_m_min	: LREAL;		// monitoring actual velocity (meter/min)
	lengthAtVelMax		: LREAL;		// monitoring: At which errorLength will setpointVel be at max? 
	
END_VAR

Tc := CycleTime;
//
// Process the position error
// 

IF Freeze THEN
	_torqueOut := ProcessValueTorqueRel;
	RETURN;
END_IF

errorLen :=  (SetPoint - ProcessValueLen);
 
(* Process deadband *)
IF Config.DeadbandLength > 0 THEN
	IF (ABS(errorLen) < (Config.DeadbandLength/2.0)) THEN
		errorLen := 0.0;
	ELSE 
		errorLen := errorLen - Signum(errorLen) * Config.DeadbandLength/2.0; 
	END_IF;
END_IF;

saveTorque(CLK := PrepareRegulator);
startTrig(CLK:=Active);

// store ProcessValueTorqueRel
IF saveTorque.Q THEN
	initialTorqueRel := ProcessValueTorqueRel;
END_IF

IF Active THEN
	// Initiatlize integrator for torque
	
	// removed, identical to next IF: 
	//IF PayoutMode AND starttrig.Q THEN
	//	It := ProcessValueTorqueRel;  //   -0.5;
	IF startTrig.Q AND IsInRun THEN
		It := initialTorqueRel; //   start the regulator with stored value
		step := 0;
	//currently as long as IsInRun is always true (see TrawlControl3), this will never run.
	ELSIF startTrig.Q AND (NOT IsInRun)  THEN
		It :=  LIMIT(0, IntegratorPresetRel, 1);  //LIMIT(-0.5, IntegratorPresetRel-0.5, 0.5);
	END_IF
	
	// set bit if haul in speed is too high
	HaulInVelocityIsOverSetpoint := SEL(ProcessValueVel <= -LimitVel,FALSE,TRUE);
	
	// limiting modes
	IF ReduceEnergyUsage THEN							// power consumed or regen too high
		step := 2; 
		velocityReduction := 0.4;
	ELSIF (ProcessValueTension  > LimitTensionMax) AND (NOT PayoutMode) THEN //too high tension (not payout)
		step := 3; 
		velocityReduction := 1;   //disabled, fixed in tension limit
	ELSIF (ProcessValueTension  < LimitTensionMin) THEN //too low tension
		step := 4; 
		velocityReduction := 1;   //disabled, fixed in tension limit
	ELSIF ProcessValueVel <= -LimitVel THEN		// haul in too fast
		step := 5; 					
		velocityReduction := 1;		// will never go too fast, limited by calculated speed ref.
	ELSIF ProcessValueVel >= LimitVel THEN		//pay out too fast
		step := 6; 
		velocityReduction := 0.50;
	ELSE										// everything's normal
		step := 1; 
		velocityReduction := 1;
	END_IF
	
	// KpVelocity: 20m error length and kp of 0.1 will give a setpointVelocity of 2 m/s or 120m/min
	// if LimitVel is active, limits and error length will be desimated accordingly limiting the setpointVelocity.
	setpointVelocity := LIMIT(-LimitVel*velocityReduction ,errorLen*config.KpVelocity*velocityReduction, LimitVel*velocityReduction);

	IF PayoutMode OR HaulInMode THEN
		IF ABS(errorLen) < 1 AND ABS(setpointVelocity) > VelStep5 THEN
			setpointVelocity := VelStep5 * signum(setpointVelocity);
		ELSIF ABS(errorLen) < 5 AND ABS(setpointVelocity) > VelStep4 THEN
			setpointVelocity := VelStep4 * signum(setpointVelocity);
		ELSIF ABS(errorLen) < 10 AND ABS(setpointVelocity) > VelStep3 THEN
			setpointVelocity := VelStep3 * signum(setpointVelocity);
		ELSIF ABS(errorLen) < 15 AND ABS(setpointVelocity) > VelStep2 THEN
			setpointVelocity := VelStep2 * signum(setpointVelocity);
		ELSIF ABS(errorLen) < 20 AND ABS(setpointVelocity) > VelStep1 THEN
			setpointVelocity := VelStep1 * signum(setpointVelocity);				
		END_IF
	END_IF	
	
	// calculate at which length the setpointVel is equal to limitVel
	// only used for monitoring
	lengthAtVelMax := (LimitVel / config.KpVelocity);
	processVel_m_min := ProcessValueVel * 60 ;
	setpointVel_m_min := setpointVelocity * 60 ;
	//
	// Tension controller -> Control velocity with torque
	//

	// The minus has to be used bc of torque has the opposite direction to velocity 
	errorVel := - (setpointVelocity - ProcessValueVel);	
	
	// If error velocity is 1 (60m) and KpTorque is 0.05 the output (Pt) will add  5% to the output signal
	
	Pt := config.KpTorque * errorVel;
	
	
	IF ABS(Config.KiTorque) <= 1E-100 THEN	// wrong parameter values
		It :=  0.0;
		deltaIt := 0.0;
	ELSE	
		// Start the check whether the new output would saturate and don't integrate when 
		// this is case
		// A KiTorque of 0.005 and errorVel of 1 (60 m/min) will increase regulator output with 0.5% per second
		deltaIt := errorVel * config.KiTorque * Tc;
		
		// don't integrate higher if we're at limitTensionMax
		IF (ProcessValueTension  > LimitTensionMax) AND deltaIt > 0 THEN
			deltaIt := 0;
		END_IF
		
		// don't integrate lower if we're at limitTensionMin
		IF (ProcessValueTension  < LimitTensionMin) AND  deltaIt < 0 THEN
			deltaIt := 0;
		END_IF
		
		// do not integrate further - probably not useful since deltaIt should be negative in this case
		IF (deltaIt > 0 AND HaulInVelocityIsOverSetpoint) THEN
			deltaIt := 0;
		END_IF
		
		tmp := Pt + It + deltaIt;
		
		// integrate when between limits
		IF ABS(tmp) <= 1  THEN		// removed 0.5 - set to '1'
			It := It + deltaIt;
		END_IF		
	END_IF

	
	_torqueOut := LIMIT(0, (Pt + It), 1);  // +0.5 removed	

ELSIF PrepareRegulator THEN
	// auto is on its way, but not active yet
	_torqueOut := initialTorqueRel ;
ELSE
	// no auto function active
	_torqueOut := ProcessValueTorqueRel;// normalized to 1
END_IF;

PROPERTY CtrlLimit : DINT
GET
CtrlLimit := Step;
END_GET
END_PROPERTY

{attribute 'TcRpcEnable'}
{attribute 'monitoring' := 'variable'}
PROPERTY ErrorPosition : LREAL
GET
ErrorPosition := errorLen;
END_GET
END_PROPERTY

{attribute 'TcRpcEnable'}
{attribute 'monitoring' := 'variable'}
PROPERTY ErrorVelocity : LREAL
GET
ErrorVelocity := errorVel;
END_GET
END_PROPERTY

{attribute 'TcRpcEnable'}
{attribute 'monitoring' := 'variable'}
PROPERTY Tension : LREAL
GET
Tension := TorqueOut;
END_GET
END_PROPERTY

PROPERTY TorqueOut : LREAL
GET
TorqueOut := _torqueOut;
END_GET
END_PROPERTY

PROPERTY VelocitySetpoint : LREAL
GET
VelocitySetpoint := setpointVelocity;
END_GET
END_PROPERTY

END_FUNCTION_BLOCK

// PID/PIDController
(*
Purpose
=======
This is a PID controller with process value and setpoint as float types.

Features
========

#. Anti Windup for the integrator
#. Low pass filter for the differentiator
#. Symmetric processing to 0 of input values
#. Limiting output values 
#. Two feed forward values to support faster changes

Methods And Properties
======================
*)
{attribute 'no_explicit_call' := 'do not call this POU directly'} 
{attribute 'hide_all_locals'}
FUNCTION_BLOCK PIDController IMPLEMENTS IPIDController;

VAR
	startTrig 			: R_TRIG;
	offset 			: LREAL;
	tmp 				: LREAL;

	_Error 				: LREAL; 
	
	E 					: ARRAY[0..1] OF LREAL;
	meas					: ARRAY[0..1] OF LREAL;
	
	P 					: LREAL;
	I 					: LREAL;
	deltaI				: LREAL;
	D 					: LREAL;
	D_1					: LREAL;
	intermediateOutput 	: LREAL;
	Tc 					: LREAL;

	_out 				: LREAL;
END_VAR

{attribute 'monitoring' := 'variable'}
{attribute 'TcRpcEnable'}
PROPERTY Error : LREAL
GET
Error := _Error;
END_GET
END_PROPERTY

{attribute 'monitoring' := 'variable'}
{attribute 'TcRpcEnable'}
PROPERTY Out : LREAL
GET
Out := _out;
END_GET
END_PROPERTY

METHOD update : LREAL
VAR_INPUT
	config 				: REFERENCE TO p7type.ConfigPID;
	Active 				: BOOL;
	Setpoint 			: LREAL;
	ProcessValue 		: LREAL;
	ProcessValueFF1 	: LREAL;
	ProcessValueFF2 	: LREAL;	
	LowerBoundary 		: LREAL;
	UpperBoundary 		: LREAL;
	CycleTime			: LREAL;
END_VAR
{warning disable C0371}
Tc := CycleTime;

startTrig(CLK:=Active);

_Error := SetPoint - ProcessValue;
 
E[1] := E[0];
E[0] := _Error; 


meas[1] := meas[0];
meas[0] := ProcessValue;

(* Process deadband *)
IF Config.Deadband > 0 THEN
	IF (ABS(E[0]) < (Config.Deadband/2.0)) THEN
		E[0] := 0.0;
		D_1 := 0;
	ELSE 
		E[0] := E[0] - Signum(E[0]) * Config.Deadband/2.0; 
	END_IF;
END_IF;

_Error := E[0];

IF Active THEN
	IF startTrig.Q  THEN
		offset := (upperBoundary - lowerBoundary)/2.0 + lowerBoundary;
		IF Config.InitializeIntegrator THEN
			// Output initializing 
			I := Config.IntegratorInit * (upperBoundary - lowerBoundary) + LowerBoundary;
		ELSE
			I := 0.0;
		END_IF
	END_IF
		
	IF ABS(config.Kd) > 0 THEN
		D := -(2.0 * config.Kd * (meas[0] - meas[1])) + (2.0 * config.Tau - Tc) * D_1 / (2.0 * config.Tau + Tc);
		D_1 := D;
	ELSE
		D_1 := 0;
		D := 0;
	END_IF
	
	P := E[0] * config.Kp;
	
	IF ABS(Config.Ki) <= 1E-100 THEN
		I := 0.0;
	ELSE
		// Start the check whether the new output would saturate and don't integrate when 
		// this is case
		deltaI := E[0] * config.Ki * Tc;	
		tmp := P + D + I + deltaI  + Config.Kf1 * ProcessValueFF1 + Config.Kf2 * ProcessValueFF2;
		IF tmp = LIMIT(lowerBoundary-offset, tmp, upperBoundary-offset) THEN
			I := LIMIT(lowerBoundary-offset, I + deltaI, upperBoundary-offset);
		END_IF
	END_IF

	tmp := P + D + I + Config.Kf1 * ProcessValueFF1 + Config.Kf2 * ProcessValueFF2;
	
	intermediateOutput := LIMIT(LowerBoundary - offset, tmp,  UpperBoundary - offset);
	
	_out := intermediateOutput + offset;	
ELSE
	_out := config.NullValue;
END_IF;
	
update := _out;
END_METHOD

END_FUNCTION_BLOCK

// PID/PIDController2P
(*
Purpose
=======
This is a PID controller with process value and setpoint as float types, 
but with 2 parameter sets. Parameter set 1 for an error value >= 0 and the another
parameter set for an error value < 0
  

Features
========

#. Anti Windup for the integrator
#. Low pass filter for the differentiator
#. Symmetric processing to 0 of input values
#. Limiting output values 
#. Two feed forward values to support faster changes

Methods And Properties
======================
*)
{attribute 'no_explicit_call' := 'do not call this POU directly'} 
{attribute 'hide_all_locals'}
FUNCTION_BLOCK PIDController2P IMPLEMENTS IPID2DController;

VAR
	startTrig 			: R_TRIG;
	offset 				: LREAL;
	tmp 				: LREAL;

	_Error 				: LREAL; 
	
	E 					: ARRAY[0..1] OF LREAL;
	meas				: ARRAY[0..1] OF LREAL;
	
	P 					: LREAL;
	I 					: LREAL;
	deltaI				: LREAL;
	D 					: LREAL;
	D_1					: LREAL;
	intermediateOutput	: LREAL;
	Tc 					: LREAL;

	_out 				: LREAL;
END_VAR

{attribute 'monitoring' := 'variable'}
{attribute 'TcRpcEnable'}
PROPERTY Error : LREAL
GET
Error := _Error;
END_GET
END_PROPERTY

{attribute 'monitoring' := 'variable'}
{attribute 'TcRpcEnable'}
PROPERTY Out : LREAL
GET
Out := _out;
END_GET
END_PROPERTY

METHOD update : LREAL
VAR_INPUT
	config 				: REFERENCE TO p7type.ConfigPID2P;
	Active 				: BOOL;
	Setpoint 			: LREAL;
	ProcessValue 		: LREAL;
	ProcessValueFF1 	: LREAL;
	ProcessValueFF2 	: LREAL;	
	LowerBoundary 		: LREAL;
	UpperBoundary 		: LREAL;
	CycleTime			: LREAL;
END_VAR
VAR_INST
	tKp, tKd, tKi, tKf1, tKf2	: LREAL;
END_VAR
{warning disable C0371}
Tc := CycleTime;

_Error := SetPoint - ProcessValue;

IF _Error >= 0.0 THEN
	tKp := config.Kp;
	tKi := config.Ki;
	tKd := config.Kd;
	tKf1 := config.Kf1;
	tKf2 := config.Kf2;
ELSE
	tKp := config.Kp2;
	tKi := config.Ki2;
	tKd := config.Kd2;
	tKf1 := config.Kf12;
	tKf2 := config.Kf22;
END_IF

Tc := CycleTime;

startTrig(CLK:=Active);

E[1] := E[0];
E[0] := _Error;


meas[1] := meas[0];
meas[0] := ProcessValue;

(* Process deadband *)
IF Config.Deadband > 0 THEN
	IF (ABS(E[0]) < (Config.Deadband/2.0)) THEN
		E[0] := 0.0;
		D_1 := 0;
	ELSE 
		E[0] := E[0] - Signum(E[0]) * Config.Deadband/2.0; 
	END_IF;
END_IF;

_Error := E[0];

IF Active THEN
	IF startTrig.Q  THEN
		offset := (upperBoundary - lowerBoundary)/2.0 + lowerBoundary;
		IF Config.InitializeIntegrator THEN
			// Output initializing 
			I := Config.IntegratorInit * (upperBoundary - lowerBoundary) + LowerBoundary;
		ELSE
			I := 0.0;
		END_IF
	END_IF
		
	IF ABS(config.Kd) > 0 THEN
		D := -(2.0 * tKd * (meas[0] - meas[1])) + (2.0 * config.Tau - Tc) * D_1 / (2.0 * config.Tau + Tc);
		D_1 := D;
	ELSE
		D_1 := 0;
		D := 0;
	END_IF

	P := E[0] * tKp;

	IF ABS(tKi) <= 1E-100 THEN
		I := 0.0;
	ELSE
		// Start the check whether the new output would saturate and don't integrate when 
		// this is case
		deltaI := E[0] * tKi * Tc;	
		tmp := P + D + I + deltaI  + tKf1 * ProcessValueFF1 + tKf2 * ProcessValueFF2;
		IF tmp = LIMIT(lowerBoundary-offset, tmp, upperBoundary-offset) THEN
			I := LIMIT(lowerBoundary-offset, I + deltaI, upperBoundary-offset);
		END_IF
	END_IF
	
	tmp := P + D + I + tKf1 * ProcessValueFF1 + tKf2 * ProcessValueFF2;
	
	intermediateOutput := LIMIT(LowerBoundary - offset, tmp,  UpperBoundary - offset);
	
	_out := intermediateOutput + offset;	
ELSE
	_out := config.NullValue;
END_IF;
	
update := _out;
END_METHOD

END_FUNCTION_BLOCK

// PID/PIDControllerLINT
(*
Purpose
=======
This is a PID controller with process value and setpoint as float types.

Features
========

#. Anti Windup for the integrator
#. Low pass filter for the differentiator
#. Symmetric processing to 0 of input values
#. Limiting output values 
#. Two feed forward values to support faster changes

Methods And Properties
======================
*)
{attribute 'no_explicit_call' := 'do not call this POU directly'} 
{attribute 'hide_all_locals'}
FUNCTION_BLOCK PIDControllerLINT;

VAR
	startTrig 			: R_TRIG;
	offset 			: LREAL;
	tmp 				: LREAL;

	_Error 				: LREAL; 
	
	E 					: ARRAY[0..1] OF LREAL;
	meas					: ARRAY[0..1] OF LINT;
	
	P 					: LREAL;
	I 					: LREAL;
	deltaI				: LREAL;
	D 					: LREAL;
	D_1					: LREAL;
	intermediateOutput 	: LREAL;
	Tc 					: LREAL;

	_out 				: LREAL;
END_VAR

{attribute 'monitoring' := 'variable'}
{attribute 'TcRpcEnable'}
PROPERTY Error : LREAL
GET
Error := _Error;
END_GET
END_PROPERTY

{attribute 'monitoring' := 'variable'}
{attribute 'TcRpcEnable'}
PROPERTY Out : LREAL
GET
Out := _out;
END_GET
END_PROPERTY

METHOD update : LREAL
VAR_INPUT
	config 				: REFERENCE TO p7type.ConfigPID;
	Active 				: BOOL;
	Setpoint 			: LINT;
	ProcessValue 		: LINT;
	ProcessValueFF1 	: LREAL;
	ProcessValueFF2 	: LREAL;	
	LowerBoundary 		: LREAL;
	UpperBoundary 		: LREAL;
	CycleTime			: LREAL;
END_VAR
VAR_INST
	dMeas 				: LREAL;
END_VAR
{warning disable C0371}
Tc := CycleTime;

startTrig(CLK:=Active);

_Error := LINT_TO_LREAL(SetPoint - ProcessValue);
 
E[1] := E[0];
E[0] := _Error; 


meas[1] := meas[0];
meas[0] := ProcessValue;

dMeas := LINT_TO_LREAL(meas[0] - meas[1]);

(* Process deadband *)
IF Config.Deadband > 0 THEN
	IF (ABS(E[0]) < (Config.Deadband/2.0)) THEN
		E[0] := 0.0;
		D_1 := 0;
	ELSE 
		E[0] := E[0] - Signum(E[0]) * Config.Deadband/2.0; 
	END_IF;
END_IF;

_Error := E[0];

IF Active THEN
	IF startTrig.Q  THEN
		offset := (upperBoundary - lowerBoundary)/2.0 + lowerBoundary;
		IF Config.InitializeIntegrator THEN
			// Output initializing 
			I := Config.IntegratorInit * (upperBoundary - lowerBoundary) + LowerBoundary;
		ELSE
			I := 0.0;
		END_IF
	END_IF
		
	IF ABS(config.Kd) > 0 THEN
		D := -(2.0 * config.Kd * dMeas) + (2.0 * config.Tau - Tc) * D_1 / (2.0 * config.Tau + Tc);
		D_1 := D;
	ELSE
		D_1 := 0;
		D := 0;
	END_IF
	
	P := E[0] * config.Kp;
	
	IF ABS(Config.Ki) <= 1E-100 THEN
		I := 0.0;
	ELSE
		// Start the check whether the new output would saturate and don't integrate when 
		// this is case
		deltaI := E[0] * config.Ki * Tc;	
		tmp := P + D + I + deltaI  + Config.Kf1 * ProcessValueFF1 + Config.Kf2 * ProcessValueFF2;
		IF tmp = LIMIT(lowerBoundary-offset, tmp, upperBoundary-offset) THEN
			I := LIMIT(lowerBoundary-offset, I + deltaI, upperBoundary-offset);
		END_IF
	END_IF

	tmp := P + D + I + Config.Kf1 * ProcessValueFF1 + Config.Kf2 * ProcessValueFF2;
	
	intermediateOutput := LIMIT(LowerBoundary - offset, tmp,  UpperBoundary - offset);
	
	_out := intermediateOutput + offset;	
ELSE
	_out := config.NullValue;
END_IF;
	
update := _out;
END_METHOD

END_FUNCTION_BLOCK

// Sensor/Fishpump/SensorBarthBase
FUNCTION_BLOCK ABSTRACT SensorBarthBase IMPLEMENTS p7type.IAnalogSensor
VAR_INPUT
	IO_In					: REFERENCE TO SensorBarthIO_In;
END_VAR
VAR
	{attribute 'hide'} 
	rvalue					: LREAL;				// Result of the pipeline			
	{attribute 'hide'} 
	_valueRaw				: LREAL;						
END_VAR

_valueRaw := io_in.input;

{attribute 'monitoring' := 'call'}
{attribute 'TcRpcEnable'}
PROPERTY Error : BOOL
GET
Error := False;
END_GET
END_PROPERTY

METHOD PROTECTED ABSTRACT processing : BOOL
END_METHOD

{attribute 'monitoring' := 'call'}
{attribute 'TcRpcEnable'}
PROPERTY Value : LREAL
GET

Value := THIS^.rvalue;
END_GET
END_PROPERTY

{attribute 'monitoring' := 'call'}
{attribute 'TcRpcEnable'}
PROPERTY ValueRaw : LREAL
GET
ValueRaw := _valueRaw;
END_GET
END_PROPERTY

END_FUNCTION_BLOCK

// Sensor/Fishpump/SensorBarthPressure
FUNCTION_BLOCK SensorBarthPressure EXTENDS SensorBarthBase IMPLEMENTS p7type.IAnalogSensor
VAR
	{attribute 'hide'} 
	pipe			: SignalPipeline;
END_VAR

SUPER^();
THIS^.processing();

METHOD PROTECTED processing : BOOL
THIS^.rvalue :=  THIS^.pipe
							.setLRealInput(WORD_TO_UINT(THIS^.io_in.input))
							.analogFilter1stDeg(0.001)
							.analogScale(190, 960, 0, 10, TRUE)
							.getAnalogValue();
END_METHOD

END_FUNCTION_BLOCK

// Sensor/Fishpump/SensorBarthTemp
(* 
This sensor class is for 4-20mA temp sensor on a EL30xx terminal with scalable range. The  output is not filtered
*)
FUNCTION_BLOCK SensorBarthTemp EXTENDS SensorBarthBase IMPLEMENTS p7type.IAnalogSensor
VAR
	{attribute 'hide'} 
	pipe			: SignalPipeline;
END_VAR

SUPER^();
THIS^.processing();

METHOD PROTECTED processing : BOOL
THIS^.rvalue :=  THIS^.pipe
							.setLRealInput(WORD_TO_UINT(THIS^.io_in.input))
							.analogScale(190, 960, -50, 150, TRUE)
							.getAnalogValue();
END_METHOD

END_FUNCTION_BLOCK

// Sensor/Fishpump/SensorBarthUnsigned
(* 
This sensor class is for 4-20mA temp sensor on a EL30xx terminal with scalable range. The  output is not filtered
*)
FUNCTION_BLOCK SensorBarthUnsigned EXTENDS SensorBarthBase IMPLEMENTS p7type.IAnalogSensor
VAR_INPUT
	ValueMax		: LREAL;
	ValueMin		: LREAL;
END_VAR
VAR
	{attribute 'hide'} 
	pipe			: SignalPipeline;
END_VAR

SUPER^();
THIS^.processing();

METHOD PROTECTED processing : BOOL
IF ABS(ValueMax-ValueMin)>=0.1 THEN
	THIS^.rvalue :=  THIS^.pipe
								.setLRealInput(WORD_TO_UINT(THIS^.io_in.input))
								.analogFilter1stDeg(0.001)
								.analogScale(190, 960, ValueMin, ValueMax, TRUE)
								.getAnalogValue();
ELSE
	THIS^.rvalue := 0.0;	
END_IF
END_METHOD

END_FUNCTION_BLOCK

// Sensor/HandlingBody/AnglePosition
(* 
This sensor class is for sensor on a EL30xx terminal with a range and offset from configvalues
*)
FUNCTION_BLOCK AnglePosition EXTENDS SensorEL30xx IMPLEMENTS IAnalogSensor
VAR
	
	{attribute 'hide'} pipe	: SignalPipeline;
END_VAR
VAR_INPUT
	config		:	REFERENCE TO  AnglePositionConfig;
END_VAR

SUPER^();
THIS^.processing();

METHOD PROTECTED processing : BOOL
THIS^.rvalue :=  THIS^.pipe
							.setLRealInput(THIS^.io_in.input)
							.analogFilter1stDeg(Config.FilterCoefficient)
							.analogScale(config.CalibratedLowerLimit, config.CalibratedUpperLimit, 0, config.MaxAngle, TRUE)
							.getAnalogValue();
END_METHOD

END_FUNCTION_BLOCK

// Sensor/SensorEL30xx
FUNCTION_BLOCK ABSTRACT SensorEL30xx IMPLEMENTS p7type.IAnalogSensor
VAR_INPUT
	IO_In					: REFERENCE TO EL30xxIO_In;
END_VAR
VAR
	{attribute 'hide'} 
	rvalue					: LREAL;				// Result of the pipeline		
	{attribute 'hide'} 
	_valueraw				: LREAL;	
END_VAR
VAR CONSTANT
	{attribute 'hide'} 
	ADC_VALUE_MAX 			: LREAL := 32767;
	ADC_VALUE_MIN 			: LREAL := -32768;
END_VAR

_valueRaw := io_in.input;

{attribute 'monitoring' := 'call'}
{attribute 'TcRpcEnable'}
PROPERTY Error : BOOL
GET
Error := False;
END_GET
END_PROPERTY

METHOD PROTECTED ABSTRACT processing : BOOL
END_METHOD

{attribute 'monitoring' := 'call'}
{attribute 'TcRpcEnable'}
PROPERTY Value : LREAL
GET

Value := THIS^.rvalue;
END_GET
END_PROPERTY

{attribute 'monitoring' := 'call'}
{attribute 'TcRpcEnable'}
PROPERTY ValueRaw : LREAL
GET
ValueRaw := _valueRaw;
END_GET
END_PROPERTY

END_FUNCTION_BLOCK

// Sensor/HandlingBody/StrokePosition
(* 
This sensor class is for sensor on a EL30xx terminal with a range of configvalues
*)
FUNCTION_BLOCK StrokePosition EXTENDS SensorEL30xx IMPLEMENTS IAnalogSensor
VAR
	{attribute 'hide'} pipe			: SignalPipeline;
	{attribute 'hide'} _Stroke		: LREAL;
	{attribute 'hide'} _Angle		: LREAL;	// In Radians
	{attribute 'hide'} _Height		: LREAL;
	{attribute 'hide'} _Length		: LREAL;
	{attribute 'hide'} _CylinderToNextBoltLength : LREAL;
END_VAR
VAR_INPUT
	config		:	REFERENCE TO  StrokePositionConfig;
END_VAR

SUPER^();
THIS^.processing();

{attribute 'monitoring' := 'call'}
{attribute 'TcRpcEnable'}
PROPERTY Angle : LREAL	// [deg]
GET
Angle := RAD_TO_DEG(_Angle);
END_GET
END_PROPERTY

{attribute 'monitoring' := 'call'}
{attribute 'TcRpcEnable'}
PROPERTY Height : LREAL
GET
Height := _Height;
END_GET
END_PROPERTY

{attribute 'monitoring' := 'call'}
{attribute 'TcRpcEnable'}
PROPERTY Length : LREAL
GET
Length := _Length;
END_GET
END_PROPERTY

METHOD PROTECTED processing : BOOL
(*for whole cylinder distance*)
THIS^.rvalue :=  THIS^.pipe	
							.setLRealInput(THIS^.io_in.input)
							.analogFilter1stDeg(Config.FilterCoefficient)
							.analogScale(config.CalibratedLowerLimit, config.CalibratedUpperLimit, config.MinStroke, config.MaxStroke, TRUE)
							.getAnalogValue();

(*for stroke distance only*)
_Stroke := THIS^.rvalue - config.MinStroke;

(*Distance to next joint needs another scaling*)
_CylinderToNextBoltLength := THIS^.pipe	
							.setLRealInput(THIS^.io_in.input)
							.analogFilter1stDeg(Config.FilterCoefficient)
							.analogScale(config.CalibratedLowerLimit, config.CalibratedUpperLimit, config.CylinderToNextJointMin, config.CylinderToNextJointMax, TRUE)
							.getAnalogValue();
							
(*Translate stroke to angle*)
IF config.BoltToCylinderBoltLength <> 0 AND config.BoltToBoltLength <> 0 THEN
	_Angle := CosineRuleKnownAllSides(
		a := config.TiltLegLength,
		b := config.BoltToBoltLength,
		c := _CylinderToNextBoltLength
	);
END_IF

(*Height*)
_Height := SIN(_Angle) * config.TiltLegLength;

(*Length*)
IF Config.InverseDirection THEN
	_Length := COS(_Angle) * config.TiltLegLength * (-1);
ELSE
	_Length := COS(_Angle) * config.TiltLegLength;	
END_IF
END_METHOD

{attribute 'monitoring' := 'call'}
{attribute 'TcRpcEnable'}
PROPERTY Stroke : LREAL
GET
Stroke := _stroke;
END_GET
END_PROPERTY

END_FUNCTION_BLOCK

// Sensor/HydPressure/HydPressure250barAA
(* 
This sensor class is for 4-20mA temp sensor on a EL30xx terminal for pressure from 0 to 250bar
*)
FUNCTION_BLOCK HydPressure250barAA EXTENDS SensorEL30xx IMPLEMENTS p7type.IAnalogSensor
VAR_INPUT
END_VAR
VAR
	{attribute 'hide'} 
	pipe			: SignalPipeline;
END_VAR

SUPER^();
THIS^.processing();

METHOD PROTECTED processing : BOOL
THIS^.rvalue :=  THIS^.pipe
							.setLRealInput(THIS^.io_in.input)
							.analogFilter1stDeg(0.01)
							.analogScale(0, THIS^.ADC_VALUE_MAX, 0, 250.0, TRUE)
							.getAnalogValue();
END_METHOD

END_FUNCTION_BLOCK

// Sensor/HydPressure/HydPressure60barAA
(* 
This sensor class is for 4-20mA temp sensor on a EL30xx terminal for pressure from 0 to 250bar
*)
FUNCTION_BLOCK HydPressure60barAA EXTENDS SensorEL30xx IMPLEMENTS p7type.IAnalogSensor
VAR_INPUT
END_VAR
VAR
	{attribute 'hide'} 
	pipe			: SignalPipeline;
END_VAR

SUPER^();
THIS^.processing();

METHOD PROTECTED processing : BOOL
THIS^.rvalue :=  THIS^.pipe
							.setLRealInput(THIS^.io_in.input)
							.analogFilter1stDeg(0.01)
							.analogScale(0, THIS^.ADC_VALUE_MAX, 0, 60.0, TRUE)
							.getAnalogValue();
END_METHOD

END_FUNCTION_BLOCK

// Sensor/OilFilter/OilFilterSensor
FUNCTION_BLOCK OilFilterSensor IMPLEMENTS p7type.IAnalogSensor;
VAR_INPUT
	OilTemperature	: LREAL;
	IO_in 			: REFERENCE TO SensorBinaryIO_in;
END_VAR
VAR
	{attribute 'hide'} 
	pipe			: SignalPipeline;
	{attribute 'hide'} 
	rvalue			: LREAL;				// Result of the pipeline
	_valueRaw		: LREAL;
END_VAR

_valueRaw := SEL(THIS^.io_in.signal, 0.0, 1.0);
THIS^.processing();

{attribute 'monitoring' := 'call'}
{attribute 'TcRpcEnable'}
PROPERTY Error : BOOL
GET
Error := FALSE;
END_GET
END_PROPERTY

METHOD PROTECTED processing : BOOL
VAR
	temp : LREAL;
END_VAR
temp := SEL(THIS^.io_in.signal, 0.0, 1.0);

temp :=  THIS^.pipe
						.setLRealInput(temp)
						.analogFilter1stDeg(Coefficient := 0.01) // tc/1s == 0.01
						.getAnalogValue();

IF OilTemperature >= 45.0 THEN						
	THIS^.rvalue := SEL(temp > 0.5, 0.0, 1.0);
ELSE
	THIS^.rvalue := 0;
END_IF
END_METHOD

{attribute 'monitoring' := 'call'}
{attribute 'TcRpcEnable'}
PROPERTY Value : LREAL
GET

Value := THIS^.rvalue;
END_GET
END_PROPERTY

{attribute 'monitoring' := 'call'}
{attribute 'TcRpcEnable'}
PROPERTY ValueRaw : LREAL
GET
ValueRaw := _valueRaw;
END_GET
END_PROPERTY

END_FUNCTION_BLOCK

// Sensor/Pressure/Pressure10barAA
(* 
This sensor class is for 4-20mA temp sensor on a EL30xx terminal with a temp range of -50C to 150C
*)
FUNCTION_BLOCK Pressure10barAA EXTENDS SensorEL30xx IMPLEMENTS p7type.IAnalogSensor
VAR
	{attribute 'hide'} 
	pipe			: SignalPipeline;
END_VAR

SUPER^();
THIS^.processing();

METHOD PROTECTED processing : BOOL
THIS^.rvalue :=  THIS^.pipe
							.setLRealInput(THIS^.io_in.input)
							.analogScale(0, THIS^.ADC_VALUE_MAX, 0, 10.0, TRUE)
							.analogFilter1stDeg(Coefficient := 0.05)
							.getAnalogValue();
END_METHOD

END_FUNCTION_BLOCK

// Sensor/Scalable/Sensor20mAA
(* 
This sensor class is for 4-20mA temp sensor on a EL30xx terminal with scalable range. The  output is not filtered
*)
FUNCTION_BLOCK Sensor20mAA EXTENDS SensorEL30xx IMPLEMENTS p7type.IAnalogSensor
VAR_INPUT
	ValueMax		: LREAL;
	ValueMin		: LREAL;
END_VAR
VAR
	{attribute 'hide'} 
	pipe			: SignalPipeline;
END_VAR

SUPER^();
THIS^.processing();

METHOD PROTECTED processing : BOOL
IF ABS(ValueMax-ValueMin)>=0.1 THEN
	THIS^.rvalue :=  THIS^.pipe
								.setLRealInput(THIS^.io_in.input)
								.analogScale(0, THIS^.ADC_VALUE_MAX, ValueMin, ValueMax, TRUE)
								.getAnalogValue();
ELSE
	THIS^.rvalue := 0.0;	
END_IF
END_METHOD

END_FUNCTION_BLOCK

// Sensor/Scalable/SensorASymRangeAA
(* 
This sensor class is for an asymetric sensor input range. The output is scalable 
*)
FUNCTION_BLOCK SensorASymRangeAA EXTENDS SensorEL30xx IMPLEMENTS p7type.IAnalogSensor
VAR_INPUT
	ValueMax		: LREAL;
	ValueMin		: LREAL;
END_VAR
VAR
	{attribute 'hide'} 
	pipe			: SignalPipeline;
END_VAR

SUPER^();
THIS^.processing();

METHOD PROTECTED processing : BOOL
IF ABS(ValueMax-ValueMin)>=0.1 THEN
	THIS^.rvalue :=  THIS^.pipe
								.setLRealInput(THIS^.io_in.input)
								.analogScale(0, THIS^.ADC_VALUE_MAX, ValueMin, ValueMax, TRUE)
								.getAnalogValue();
ELSE
	THIS^.rvalue := 0.0;	
END_IF
END_METHOD

END_FUNCTION_BLOCK

// Sensor/Scalable/SensorSymRange
(* 
This sensor class is for a symetric input range. The output is scalable 
*)
FUNCTION_BLOCK SensorSymRange EXTENDS SensorEL30xx IMPLEMENTS p7type.IAnalogSensor
VAR_INPUT
	ValueRawMin		: LREAL;
	ValueRawMax		: LREAL;
	ValueMax		: LREAL;
	ValueMin		: LREAL;
END_VAR
VAR
	{attribute 'hide'} 
	pipe			: SignalPipeline;
END_VAR

SUPER^();
THIS^.processing();

METHOD PROTECTED processing : BOOL
IF ABS(ValueMax-ValueMin)>=0.1 THEN
	THIS^.rvalue :=  THIS^.pipe
								.setLRealInput(THIS^.io_in.input)
								.analogScale(ValueRawMin, ValueRawMax, ValueMin, ValueMax, TRUE)
								.getAnalogValue();
ELSE
	THIS^.rvalue := 0.0;	
END_IF
END_METHOD

END_FUNCTION_BLOCK

// Sensor/Scalable/SensorSymRangeAA
(* 
This sensor class is for a symetric input range. The output is scalable 
*)
FUNCTION_BLOCK SensorSymRangeAA EXTENDS SensorEL30xx IMPLEMENTS p7type.IAnalogSensor
VAR_INPUT
	ValueMax		: LREAL;
	ValueMin		: LREAL;
END_VAR
VAR
	{attribute 'hide'} 
	pipe			: SignalPipeline;
END_VAR

SUPER^();
THIS^.processing();

METHOD PROTECTED processing : BOOL
IF ABS(ValueMax-ValueMin)>=0.1 THEN
	THIS^.rvalue :=  THIS^.pipe
								.setLRealInput(THIS^.io_in.input)
								.analogScale(THIS^.ADC_VALUE_MIN, THIS^.ADC_VALUE_MAX, ValueMin, ValueMax, TRUE)
								.getAnalogValue();
ELSE
	THIS^.rvalue := 0.0;	
END_IF
END_METHOD

END_FUNCTION_BLOCK

// Sensor/Temperature/TempSensorAB
(* 
This sensor class is for 4-20mA temp sensor on a EL30xx terminal with a temp range of -50C to 150C
*)
FUNCTION_BLOCK TempSensorAB EXTENDS SensorEL30xx IMPLEMENTS p7type.IAnalogSensor
VAR
	{attribute 'hide'} 
	pipe			: SignalPipeline;
END_VAR

SUPER^();
THIS^.processing();

METHOD PROTECTED processing : BOOL
THIS^.rvalue :=  THIS^.pipe
							.setLRealInput(THIS^.io_in.input)
							.analogScale(0, THIS^.ADC_VALUE_MAX, 0.0, 100.0, TRUE)
							.analogFilter1stDeg(Coefficient := 0.001)
							.getAnalogValue();
END_METHOD

END_FUNCTION_BLOCK

// Sensor/Temperature/TempSensorAC
(* 
This sensor class is for 4-20mA temp sensor on a EL30xx terminal with a temp range of -50C to 150C
*)
FUNCTION_BLOCK TempSensorAC EXTENDS SensorEL30xx IMPLEMENTS p7type.IAnalogSensor
VAR
	{attribute 'hide'} 
	pipe			: SignalPipeline;
END_VAR

SUPER^();
THIS^.processing();

METHOD PROTECTED processing : BOOL
THIS^.rvalue :=  THIS^.pipe
							.setLRealInput(THIS^.io_in.input)
							.analogScale(0, THIS^.ADC_VALUE_MAX, -50.0, 130.0, TRUE)
							.analogFilter1stDeg(Coefficient := 0.001)
							.getAnalogValue();
END_METHOD

END_FUNCTION_BLOCK

// Sensor/Temperature/TempSensorAA
(* 
This sensor class is for 4-20mA temp sensor on a EL30xx terminal with a temp range of -50C to 150C
*)
FUNCTION_BLOCK TempSensorAA EXTENDS SensorEL30xx IMPLEMENTS p7type.IAnalogSensor
VAR
	{attribute 'hide'} 
	pipe			: SignalPipeline;
END_VAR

SUPER^();
THIS^.processing();

METHOD PROTECTED processing : BOOL
THIS^.rvalue :=  THIS^.pipe
							.setLRealInput(THIS^.io_in.input)
							.analogScale(0, THIS^.ADC_VALUE_MAX, -50.0, 150.0, TRUE)
							.analogFilter1stDeg(Coefficient := 0.001)
							.getAnalogValue();
END_METHOD

END_FUNCTION_BLOCK

// Sensor/DummySensor
FUNCTION_BLOCK DummySensor IMPLEMENTS IAnalogSensor

{attribute 'monitoring' := 'call'}
{attribute 'TcRpcEnable'}
PROPERTY Error : BOOL
GET
Error := FALSE;
END_GET
END_PROPERTY

{attribute 'monitoring' := 'call'}
{attribute 'TcRpcEnable'}
PROPERTY Value : LREAL
GET

Value := 0.0;
END_GET
END_PROPERTY

{attribute 'monitoring' := 'call'}
{attribute 'TcRpcEnable'}
PROPERTY ValueRaw : LREAL
GET
END_GET
END_PROPERTY

END_FUNCTION_BLOCK

// SignalClassifier/SignalClassGTEQ
{attribute 'hide_all_locals'}
FUNCTION_BLOCK SignalClassGTEQ EXTENDS SignalPipeline
VAR
	sensor				: IAnalogSensorBase;
	signalLimit			: LREAL;
	signalHysteresis	: LREAL; 	
	filterCoefficient	: LREAL;
	minTime				: TIME;
	bvalue				: BOOL;
END_VAR

METHOD PROTECTED processing : BOOL
THIS^.bvalue := THIS^
				.setLRealInput(THIS^.sensor.Value)
				.analogFilter1stDeg(THIS^.filterCoefficient) 
				.testGreaterOrEqual(THIS^.signalLimit - THIS^.signalHysteresis/2.0, THIS^.signalHysteresis, FALSE)
				.boolTestTimeSpan(TimeSpan := THIS^.minTime)
				.getBinaryValue();
END_METHOD

PROPERTY Signal : BOOL
GET
Signal := THIS^.bvalue;
END_GET
END_PROPERTY

METHOD update : BOOL
VAR_INPUT
	Sensor				: IAnalogSensorBase;
	SignalLimit			: LREAL;
	SignalHysteresis	: LREAL; 
	FilterCoefficient	: LREAL;
	MinTime				: TIME;
END_VAR
THIS^.sensor 			:= Sensor; 
THIS^.signalLimit 		:= SignalLimit;
THIS^.signalHysteresis 	:= SignalHysteresis;
THIS^.filterCoefficient := FilterCoefficient;
THIS^.minTime			:= MinTime;
THIS^.processing();
END_METHOD

END_FUNCTION_BLOCK

// SignalClassifier/SignalClassLTEQ
{attribute 'hide_all_locals'}
FUNCTION_BLOCK SignalClassLTEQ EXTENDS SignalPipeline
VAR
	sensor				: IAnalogSensor;
	signalLimit			: LREAL;
	signalHysteresis	: LREAL; 	
	filterCoefficient	: LREAL;
	minTime				: TIME;
	bvalue				: BOOL;
END_VAR

METHOD PROTECTED processing : BOOL
THIS^.bvalue := THIS^
				.setLRealInput(THIS^.sensor.Value)
				.analogFilter1stDeg(THIS^.filterCoefficient) 
				.testLessOrEqual(THIS^.signalLimit + THIS^.signalHysteresis/2.0, THIS^.signalHysteresis, FALSE)
				.boolTestTimeSpan(TimeSpan := THIS^.minTime)
				.getBinaryValue();
END_METHOD

PROPERTY Signal : BOOL
GET
Signal := THIS^.bvalue;
END_GET
END_PROPERTY

METHOD update : bool
VAR_INPUT
	Sensor				: IAnalogSensor;
	SignalLimit			: LREAL;
	SignalHysteresis	: LREAL; 
	FilterCoefficient	: LREAL;
	MinTime				: TIME;
END_VAR
THIS^.sensor 			:= Sensor; 
THIS^.signalLimit 		:= SignalLimit;
THIS^.signalHysteresis 	:= SignalHysteresis;
THIS^.filterCoefficient := FilterCoefficient;
THIS^.minTime			:= MinTime;
THIS^.processing();
END_METHOD

END_FUNCTION_BLOCK

// SignalProcessing/Filter1stDegEx
(*
Purpose
=======
This is a 1st deg filter class. The coeffcient has a range from 0..1 and is limited automagically by this class


Methods And Properties
======================
*)
{attribute 'hide_all_locals'}
FUNCTION_BLOCK Filter1stDegEx
VAR_INPUT
	Value 			: LREAL;
	Coefficient  	: LREAL;
END_VAR
VAR_OUTPUT
	Out 			: LREAL; 
END_VAR
VAR
	value_1 		: LREAL;
	value_0			: LREAL;
	CoefficientCopy : LREAL;
END_VAR


CoefficientCopy := LIMIT(0.0, Coefficient, 1.0);
value_0 := Value * CoefficientCopy + (1.0 - CoefficientCopy) * value_1; 

value_1 := value_0;

Out 	:= value_0;

METHOD reset : BOOL
value_0 := 0;
value_1 := 0;
END_METHOD

END_FUNCTION_BLOCK

// SignalProcessing/TwoSideTest
(*
Purpose
=======
This class is a hysteresis test for a band. Ther borders have a hysteresis.
The output is 1 when value is greater than max band value and -1 , when output is less
then min band value. 


Methods And Properties
======================
*)
{attribute 'hide_all_locals'}
FUNCTION_BLOCK TwoSideTest
VAR_INPUT
	BandCenter		: LREAL;  // Band center 
	BandWidth		: LREAL;  // Band width
	Hysteresis 		: LREAL;  // Hysteresis
	Value			: LREAL;
END_VAR
VAR_OUTPUT
	Out				: LREAL;
END_VAR
VAR
	state : SwitchHysteresisSM;
END_VAR


CASE state OF 
	SwitchHysteresisSM.START:
		state := SwitchHysteresisSM.IDLE; 
		
	SwitchHysteresisSM.IDLE:
		IF Value >= BandCenter + ABS(BandWidth/2.0) + ABS(Hysteresis/2.0) THEN
			state := SwitchHysteresisSM.BANDUP;
		ELSIF  Value <= BandCenter - ABS(BandWidth/2.0) - ABS(Hysteresis/2.0) THEN
			state := SwitchHysteresisSM.BANDDOWN;
		END_IF
				
	SwitchHysteresisSM.BANDUP:
		IF Value <= BandCenter + ABS(BandWidth/2.0) - ABS(Hysteresis/2.0) THEN
			state := SwitchHysteresisSM.IDLE;
		END_IF
		
	SwitchHysteresisSM.BANDDOWN:
		IF Value >= BandCenter - ABS(BandWidth/2.0) + ABS(Hysteresis/2.0) THEN
			state := SwitchHysteresisSM.IDLE;
		END_IF
		
	ELSE
		state := SwitchHysteresisSM.START;
END_CASE

IF state = SwitchHysteresisSM.BANDUP THEN
	Out := 1;
ELSIF state = SwitchHysteresisSM.BANDDOWN THEN
	Out := -1;
ELSE
	Out := 0;	
END_IF

END_FUNCTION_BLOCK

// Signals/OneShotSignal
{attribute 'no_explicit_call' := 'do not call this POU directly'} 
FUNCTION_BLOCK OneShotSignal
VAR
	flag : BOOL;
END_VAR

METHOD Get : BOOL
VAR_INPUT
END_VAR
Get 	:= flag;
flag 	:= FALSE;
END_METHOD

METHOD Set : BOOL
VAR_INPUT
END_VAR
flag := TRUE;
END_METHOD

END_FUNCTION_BLOCK

// Signals/OneShotSignalInt
{attribute 'no_explicit_call' := 'do not call this POU directly'} 
FUNCTION_BLOCK OneShotSignalInt
VAR
	_value : INT;
END_VAR

METHOD Get : INT
VAR_INPUT
END_VAR
Get 	:= _value;
_value 	:= -32768;
END_METHOD

METHOD Set : INT
VAR_INPUT
	Value : INT;
END_VAR
_value := Value;
END_METHOD

END_FUNCTION_BLOCK

// TimingGenerators/CycleGenerator
(*
Purpose
=======
This class outputs a pulse every x sec and takes into account the initialisation of
a TON timer. 

Caveats
=======
The used time period has to be >= 4 x cycle time and the period is limited to 1s

Methods And Properties
======================
*)
{attribute 'no_explicit_call' := 'do not call this POU directly'} 
{attribute 'hide_all_locals'}
FUNCTION_BLOCK CycleGenerator
VAR
	timer 			: TON;
END_VAR

PROPERTY Q : BOOL
GET
Q := timer.Q;
END_GET
END_PROPERTY

METHOD update : BOOL
VAR_INPUT
	In : TIME; // Time 
	PLCTask_CycleTime : TIME;
END_VAR
VAR_INST
	Ts 		: TIME := p7type.CycleTime_Task0;
END_VAR

timer(In:=NOT timer.Q, PT:= In - (Ts * 2));

update := timer.Q;
END_METHOD

END_FUNCTION_BLOCK

// TimingGenerators/CycleTimer
(*
	This FB is implementing a cycle timer as a tool to secure a minium amount of cycles in the 
	communication between statemachines.
*)
{attribute 'hide_all_locals'}
FUNCTION_BLOCK CycleTimer
VAR_INPUT
IN 		: BOOL;
Cycles 	: UDINT;
END_VAR
VAR_OUTPUT
	ET	: UDINT;
	Q 	: BOOL;
END_VAR
VAR
	trigStart : R_TRIG;
END_VAR


trigStart(CLK:=IN);

IF trigStart.Q THEN
	ET := Cycles;
ELSE
	IF ET <> 0 THEN
		ET := ET - 1;
	END_IF
END_IF

Q := ET = 0;

END_FUNCTION_BLOCK

// UnitConversion/UnitConverter
FUNCTION_BLOCK UnitConverter
VAR CONSTANT
	// Length Units
	{attribute 'hide'} _meters : LREAL := 1.0;
	{attribute 'hide'} _feet : LREAL := 3.28084;
	{attribute 'hide'} _fathoms : LREAL := 0.546807;
	
	//Tension units
	{attribute 'hide'} _tonnesMetric : LREAL := 0.001;
	{attribute 'hide'} _tonnesImperial : LREAL := 0.000984207;
	{attribute 'hide'} _pounds : LREAL := 2.20462;
	{attribute 'hide'} _kilos : LREAL := 1.0;

	// Velocity units
	{attribute 'hide'} _mPerSecond : LREAL := 1.0;
	{attribute 'hide'} _mPerMinute : LREAL := 60.0;
	{attribute 'hide'} _feetPerMinute : LREAL := 196.85;
	{attribute 'hide'} _fathomsPerMinute  : LREAL := 32.8084;
	
	{attribute 'hide'} _meterString : STRING := 'm';
	{attribute 'hide'} _feetString : STRING := 'ft';
	{attribute 'hide'} _fathomsString : STRING := 'ftm';

	//Velocity string
	{attribute 'hide'} _mPerSecondString : STRING := 'm/s';
	{attribute 'hide'} _mPerMinuteString : STRING := 'm/Min';
	{attribute 'hide'} _feetPerMinuteString : STRING := 'Ft/Min';
	{attribute 'hide'} _fathomsPerMinuteString : STRING := 'Ftm/Min';

	//Tension String
	{attribute 'hide'} _tonnesMetricString : STRING := 't';
	{attribute 'hide'} _tonnesImperialString : STRING := 't';
	{attribute 'hide'} _poundsString : STRING := 'lbs';
	{attribute 'hide'} _kilosString : STRING := 'kg';
	
END_VAR

METHOD getLengthUnit : STRING
VAR_INPUT
	Unit : LengthUnits;
END_VAR
CASE Unit OF
	LengthUnits.METER:
		getLengthUnit := _meterString;
		
	LengthUnits.FEET:
		getLengthUnit := _feetString;
		
	LengthUnits.FATHOM:
		getLengthUnit := _fathomsString;
END_CASE
END_METHOD

METHOD getTensionUnit : STRING
VAR_INPUT
	Unit : TensionUnits;
END_VAR
CASE Unit OF
	
	TensionUnits.TON_METRIC:
		getTensionUnit := _tonnesMetricString;
		
	TensionUnits.TON_IMPERIAL:
		getTensionUnit := _tonnesImperialString;
		
	TensionUnits.POUND:
		getTensionUnit := _poundsString;
		
	TensionUnits.KILO:
		getTensionUnit := _kilosString;	
END_CASE
END_METHOD

METHOD getVelocityUnit : STRING
VAR_INPUT
	Unit : VelocityUnits;
END_VAR
CASE Unit OF
	
	VelocityUnits.METER_PER_SEC:
		getVelocityUnit:= _mPerSecondString;
		
	VelocityUnits.METER_PER_MIN:
		getVelocityUnit := _mPerMinuteString;
		
	VelocityUnits.FEET_PER_MIN:
		getVelocityUnit := _feetPerMinuteString;
	
	VelocityUnits.FATHOM_PER_MIN:
		getVelocityUnit := _fathomsPerMinuteString;
		
END_CASE
END_METHOD

METHOD kgToUnit : LREAL
VAR_INPUT
	Unit 	: TensionUnits;
	Value 	: LREAL;
END_VAR
CASE Unit OF	
	TensionUnits.TON_METRIC:
		kgToUnit := Value * _tonnesMetric;
		
	TensionUnits.TON_IMPERIAL:
		kgToUnit := Value * _tonnesImperial;
		
	TensionUnits.POUND:
		kgToUnit := Value * _pounds;
		
	TensionUnits.KILO:
		kgToUnit := Value;
END_CASE
END_METHOD

METHOD meterToUnit : LREAL
VAR_INPUT
	Unit 	: LengthUnits;
	Value	: LREAL;
END_VAR
CASE Unit OF
	
	LengthUnits.METER:
		meterToUnit := Value;
		
	LengthUnits.FEET:
		meterToUnit := _feet * Value;
		
	LengthUnits.FATHOM:
		meterToUnit := _fathoms * Value;
		
END_CASE
END_METHOD

METHOD MSToUnit : LREAL
VAR_INPUT
	Unit : VelocityUnits;
	Value : LREAL;
END_VAR
CASE Unit OF
	
	VelocityUnits.METER_PER_SEC:
		MSToUnit := _mPerSecond;
		
	VelocityUnits.METER_PER_MIN:
		MSToUnit := Value * _mPerMinute;
		
	VelocityUnits.FEET_PER_MIN:
		MSToUnit := Value * _feetPerMinute;
	
	VelocityUnits.FATHOM_PER_MIN:
		MSToUnit := Value * _fathomsPerMinute;
		
END_CASE
END_METHOD

METHOD unitToKg : LREAL
VAR_INPUT
	Unit 	: TensionUnits;
	Value 	: LREAL;
END_VAR
CASE Unit OF
	TensionUnits.TON_METRIC:
		unitToKg := Value / _tonnesMetric;
		
	TensionUnits.TON_IMPERIAL:
		unitToKg := Value / _tonnesImperial;
		
	TensionUnits.POUND:
		unitToKg := Value / _pounds;
		
	TensionUnits.KILO:
		unitToKg := Value;
END_CASE
END_METHOD

METHOD unitToMeter : LREAL
VAR_INPUT
	Unit 	: LengthUnits;
	Value	: LREAL;
END_VAR
CASE Unit OF
	
	LengthUnits.METER:
		unitToMeter := Value;
		
	LengthUnits.FEET:
		unitToMeter := Value/_feet;
		
	LengthUnits.FATHOM:
		unitToMeter := Value/_fathoms;
		
END_CASE
END_METHOD

METHOD unitToMS : LREAL
VAR_INPUT
	Unit : VelocityUnits;
	Value : LREAL;
END_VAR
CASE Unit OF
	
	VelocityUnits.METER_PER_SEC:
		unitToMS := _mPerSecond;
		
	VelocityUnits.METER_PER_MIN:
		unitToMS := Value / _mPerMinute;
		
	VelocityUnits.FEET_PER_MIN:
		unitToMS := Value / _feetPerMinute;
	
	VelocityUnits.FATHOM_PER_MIN:
		unitToMS := Value / _fathomsPerMinute;
		
END_CASE
END_METHOD

END_FUNCTION_BLOCK
